(* IEC 61131-3 sources: Mizera_Tube/Plc (part 17) *)

*******************************************************************************
*   @@@ RICERCA BLOCCO
*******************************************************************************

LD   BUP_BLKSRC_PAGE               ** User in block search page
ST   GESTCH0.xBlkSearch

LD   %PLCFLAGS.1
ST   GESTCH0.xIntBlkSrc    * Forzam. esec. ricerca blocco interna

LD   %PlcOp0.2                     ** DryRun
ST   GESTCH0.xSpeedDryRunEnab ** Ab. velocita' di Dry Run (disabled in cnc.plc)

LD   %PLCFLAGS.0
ST   GESTCH0.xOverstore  * Ab. overstore dopo ricerca blocco (provv.)

LD   CondHoldCN0                   ** Condizioni richiesta hold canale 0
AND  PRGRUN_CN0                    ** M0.0 cn0.rc8.0  Programma in corso
ANDN BCO_CUSTOM_BOOT               ** rc8.18 Ciclo $BOOT in corso
ANDN BCO_CUSTOM_RESET              ** rc8.20 Ciclo $RESET in corso
ANDN PRGSTOP_CN0                   ** (cn0.rc8.1)  Programma interrotto CN0
ST   GESTCH0.xHold                * comando Hold al canale (esterno)

LD   Res_Ch0                       ** (gPlc25.3) reset channel 0
ST   GESTCH0.xReset               * comando RESET al canale (esterno)

CAL  FTRIG_POT (CLK:=Pon)          ** PON
CAL  TP_FTRIG_POT(IN:=FTRIG_POT.Q,PT:=300)

LD   %cn0.rc8.0
AND (
LD   bevAngleHead1_calc1                  * (C154) head 1 bevel angle
GE   70000
)
AND  %uvHeads0.uvhCommand[0].1          * UVH_COMMAND_PLC_VRTC_HANDLING
S    alarm_tool_surface

LD   %cn0.rc8.0
AND (
LD   %cn0.rc18                      * CO_ERRCODE
EQ   428                            * motion command error
)
S    alarm_motion_cmd_err

LD   Pul_Reset                     ** (gPlc0.3)Reset pushbutton
R    alarm_tool_surface
R    alarm_motion_cmd_err

LD   alarm_tool_surface
ST   %PLCerr4.0

LD   alarm_motion_cmd_err
ST   %PLCerr4.1

* todo CAL  RTRIG_TIPTOUCH(CLK:=%PLCerr5.4)

LD   Pul_Reset                     ** (gPlc0.3)Reset pushbutton
OR   Pul_Stop                      ** (gPlc0.2)Stop pushbutton
AND  ch0_in_ref                    ** channel 0 in ref
OR   EMER_GEN                      ** M0.10 Emergenza generale
***OR   LsrVrtcFcSoftware             ** (LsPlc0.31)Intervento Fc Sofware in lavorazione Laser
OR   TP_FTRIG_POT.Q
OR (
LD   %vrtc1.VrdwStatRegister1.2     * Upper mandatory position limit reached
OR   %vrtc1.VrdwStatRegister1.3     * Lower mandatory position limit reached
AND  %vrtc1.VrdwCtrlRegister0.1
)
* todo OR   RTRIG_TIPTOUCH.Q
OR   alarm_tool_surface
OR   alarm_motion_cmd_err
OR   Pul_Reset_EMERG                * Tasto RESET premuto per pi?di 4 secondi
ST   GESTCH0.xEmer

LD   ChannelFeedrate               ** feedrate for channel
ST   GESTCH0.xOverride
ST   AxesOverride

**********************************************************************
* Limitazione 10% to 100% in case of following supports in descending
**********************************************************************
LD   EnVSuppFeedRec
JMPCN STATE_EN_VSREC
LD   GESTCH0.xOverride
MULDIV(M=VSuppFeedReduction,D=1000)
ST   GESTCH0.xOverride
STATE_EN_VSREC:
**********************************************************************

CAL  GESTCH0

*******************************************************************************
*   @@@ RICERCA BLOCCO
*******************************************************************************
LD   GESTCH0.yBlkSearch
ST   BLKSRC_RUN                    ** Ricerca blocco in corso

LD   GESTCH0.yBlkSrcEnded * ricerca blocco terminata
ST   BLKSRC_END                    ** Ricerca blocco terminata

LD   0
ST   %cn0.BlkSearch.MskMoveA

LD   16#32
ST   %cn0.BlkSearch.Option

LD   BUP_BLKSRCPOINT               ** ui16.31 Ricerca blocco su punto intermedio
JMPCN INTPOINT

LD   16#72
ST   %cn0.BlkSearch.Option

INTPOINT:
LD   -1
ST   %ui6           ** Non generare M su overstore automatico
ST   %ui7           ** Non generare S/T su overstore automatico

***********************************************
* Gestione Informazioni per ripresa lavorazione
***********************************************

LD   Pul_Start                     ** (gPlc0.1)Start pushbutton
AND  ch0_in_aut                    ** channel 0 in aut
ANDN ExeAuxMode                    ** (gPlc0.29)Esecuzione ausiliaria 1000.PGM
S    MEM_INTPROG                   ** R15.0 Mem. programma valido per ripresa pezzo

LD   M30_CN0                       ** M0.13 M30:EndProgram CN0
ANDN ExeAuxMode                    ** (gPlc0.29)Esecuzione ausiliaria 1000.PGM
OR   BUP_PROGSEL                   ** ui16.30 Impulso selezione programma
R    MEM_INTPROG                   ** R15.0 Mem. programma valido per ripresa pezzo

* Lettura dati correnti durante esecuzione programma

LD   %cn0.rc8.0          * Programma in corso canale 0
ANDN %cn0.rc0.0          * Reset NC
***ANDN KeyStop_Tp          ** Stop level
ANDN %cn0.rc8.1          * rc8.1  Programma interrotto
ANDN %cn0.rc8.8
ANDN ExeAuxMode                    ** (gPlc0.29)Esecuzione ausiliaria 1000.PGM
JMPCN READ

LD   %cn0.lev0.curline
ST   CURRENT_LINE                  ** Numero riga corrente del part program in esecuzione

*******************************************
*   Calcola la posizione del TCP sul piano
*   della macchina
*******************************************
LDN  Gest5Ax                        ** (gPlc0.0)Gestione MAcchina 5 assi
JMPC Normal

LD   %ax0.ra54          ** X TCP
ST   locX                          ** Used in block search (ricerca blocco)

LD   %ax1.ra54          ** Y TCP
ST   locY                          ** Used in block search (ricerca blocco)

LD   %cn0.mat.sts0
EQ   16#B
JMPCN identity

LD   locX                          ** Used in block search (ricerca blocco)
DIV  100                ** DIV per problemi di overflow
MUL  %cn0.mat.a0
ADD  (
LD   locY                          ** Used in block search (ricerca blocco)
DIV  100
MUL  %cn0.mat.a1
)
DIV  10
ADD  (
LD   %cn0.mat.a3
DIV  1000
)
ST   XactualQta                    ** X actual quota Used in block search (ricerca blocco)

LD   locX                          ** Used in block search (ricerca blocco)
DIV  100                ** DIV per problemi di overflow
MUL  %cn0.mat.a4
ADD  (
LD   locY                          ** Used in block search (ricerca blocco)
DIV  100
MUL  %cn0.mat.a5
)
DIV  10
ADD  (
LD   %cn0.mat.a7
DIV  1000
)
ST   YactualQta                    ** Y actual quota Used in block search (ricerca blocco)

JMP  ComHead

identity:
LD   locX                          ** Used in block search (ricerca blocco)
ST   XactualQta                    ** X actual quota Used in block search (ricerca blocco)

LD   locY                          ** Used in block search (ricerca blocco)
ST   YactualQta                    ** Y actual quota Used in block search (ricerca blocco)

JMP  ComHead

Normal:
LD   %ax0.ra4           ** X
ST   XactualQta                    ** X actual quota Used in block search (ricerca blocco)

LD   %ax1.ra4           ** Y
ST   YactualQta                    ** Y actual quota Used in block search (ricerca blocco)

ComHead:
LD   XactualQta                    ** X actual quota Used in block search (ricerca blocco)
SUB  ORIGPRGX                      ** Origine programmata X
ST   MEM_XQUOTE                    ** R13 Memorizza quota X per collimazione ricerca blocco

LD   YactualQta                    ** Y actual quota Used in block search (ricerca blocco)
SUB  ORIGPRGY                      ** Origine programmata Y
ST   MEM_YQUOTE                    ** R14 Memorizza quota Y per collimazione ricerca blocco

READ:
* Azzera dati se programma non valido

LD   MEM_INTPROG                   ** R15.0 Mem. programma valido per ripresa pezzo
JMPC END_VALPR

LD   0
ST   CURRENT_LINE                  ** Numero riga corrente del part program in esecuzione
ST   MEM_XQUOTE                    ** R13 Memorizza quota X per collimazione ricerca blocco
ST   MEM_YQUOTE                    ** R14 Memorizza quota Y per collimazione ricerca blocco

END_VALPR:

* Passa i dati alla UI
* NB: occorre saltare l'aggiornamento nella modalita di overstore/auxcmd

LD   %cn0.rc8.26
ANDN %cn0.rc8.24
OR(
LD   %cn0.rc8.27
ANDN %cn0.rc8.25
)
JMPC OVERSTORERUN

LD   CURRENT_LINE                  ** Numero riga corrente del part program in esecuzione
*ADD  1
ST   PU_LASTLINE                   ** ui13 Ultima linea eseguita per ricerca blocco

LD   MEM_XQUOTE                    ** R13 Memorizza quota X per collimazione ricerca blocco
ST   PU_QCOLX                      ** ui2 Quota asse X collimazione ricerca blocco

LD   MEM_YQUOTE                    ** R14 Memorizza quota Y per collimazione ricerca blocco
ST   PU_QCOLY                      ** ui3 Quota asse Y collimazione ricerca blocco

OVERSTORERUN:

* Abilita quote per collimazione ricerca blocco

LD   MEM_INTPROG                   ** R15.0 Mem. programma valido per ripresa pezzo
ST   PLC_BPU_ENCOLDATA             ** ui0.31 Abilita quote per collimazione ricerca blocco

LD   PLC_BPU_ENCOLDATA             ** ui0.31 Abilita quote per collimazione ricerca blocco
ANDN PRGRUN_CN0                    ** M0.0 cn0.rc8.0  Programma in corso
ST   ResumeProgEnab                ** (gPlc25.0) Data avaiable for resume program

LD   Pul_Start                     ** (gPlc0.1)Start pushbutton
ANDN ExeAuxMode                    ** (gPlc0.29)Esecuzione ausiliaria 1000.PGM
AND  ch0_in_aut                    ** channel 0 in aut
S    BlackOut                      ** (R55.31)Interruzione per BlackOut

LD   FT_PRGRUN.Q        ** Dwn Programma in corso
OR   Pul_Reset                     ** (gPlc0.3)Reset pushbutton
OR   M30_CN0                       ** M0.13 M30:EndProgram CN0
R    BlackOut                      ** (R55.31)Interruzione per BlackOut

*******************************************************************************

LD   GESTCH0.yProgramRun * Programma in corso
ST   PRGRUN_CN0                    ** M0.0 cn0.rc8.0  Programma in corso

LD   BCO_STB_GET                   ** rc8.17 Strobe per GET resources
AND  AxStopSincGRP                 ** (gPlc13.11)Assi Fermi per sincronismo GRP[ax]
ST   BCI_ACK_GET                   ** rc0.29  ACK per GET resource

LD   GESTCH0.xRTPlus     * comando + in retrace
AND  %cn0.rc64.25        * Comando FWD Retrace
OR(
LD   GESTCH0.xRTMinus    * comando - in retrace
AND  %cn0.rc64.26        * Comando REV Retrace
)
AND  M_HOLD                        ** (gPlc19.0)Mem. Richiesta Hold
ST   Appoggio                      ** Appoggio

CAL  TOF_0(IN=Appoggio,PT=1000)    ** Appoggio

LD   TOF_0.Q
ST   RETRACERUN                    ** M0.11 Ciclo di retrace in Run

**************************
* FUNZIONI M DI SERVIZIO *
*      CANALE 0          *
**************************

LD   %rc9                * Registro funzioni M canale 0
EQ   10
AND  %rc8.4              * Strobe funzioni M canale 0
ST   M10_CN0                       ** M0.14 M10: Attiva Hold + Jog CN0

LD   %rc9                * Registro funzioni M canale 0
EQ   30
AND  %rc8.4              * Strobe funzioni M canale 0
ST   M30_CN0                       ** M0.13 M30:EndProgram CN0

LD   %rc9                * Registro funzioni M canale 0
EQ   2
AND  %rc8.4              * Strobe funzioni M canale 0
ST   M2_CN0                        ** M0.28 M2: EndProgram CN0 M2

LD   %rc9                * Registro funzioni M canale 0
EQ   32
AND  %rc8.4              * Strobe funzioni M canale 0
ST   M32TglMan                     ** M32: Attesa inizio taglio manuale

****************************************************************************************************

*** *** ***

LD   %rc9                * Registro funzioni M canale 0
EQ   600
AND  %rc8.4              * Strobe funzioni M canale 0
ST   M600_G81_84                   ** Richiesta Sblocco M40000_CN4: Richiesta Servizio per Unit_2]

CAL  TP_1(IN=M600_G81_84,PT=1000)  ** Impulso sblocco M40000

**************************
LD   %rc9                * Registro funzioni M canale 0
EQ   7000
AND  %rc8.4              * Strobe funzioni M canale 0
ST   M7000_RETR                    ** M7000: Retrace enable

LD   %rc9                * Registro funzioni M canale 0
EQ   8000
AND  %rc8.4              * Strobe funzioni M canale 0
ST   M8000_RETR                    ** M8000: Retrace disable
**************************

********************************************************************************
* DB Laser upload synchronism
********************************************************************************
*LD   %LSRPlcOp0.5                  ** Worklist mode enabled
*AND  %WlistMngt.wl_flag.0       ** Se codice DB gestito nella linea della lista di lavoro
*ORN  %LSRPlcOp0.5                  ** Worklist mode enabled
*JMPCN NoLoadDB

LD   %cn0.rc9                   ** Registro funzioni M canale 0
EQ   1000
AND  %cn0.rc8.4                 ** Strobe funzioni M canale 0
OR   isoLoadRecord                 ** (LsIso10.3) Load database record with Block search in run
ST   Up_Load_DB                    ** upload DB request

CAL  RTRIG_CAR_DB(CLK:=Up_Load_DB) ** Trig on upload DB request

LD   RTRIG_CAR_DB.Q
S    UpLoad_DB_Laser               ** (LsPlc0.0 )Comando Caricamento DataBase Laser

*NoLoadDB:
LD   FeedbackDBloaded              ** (LsGui1.0) upload DB request
OR   Pul_Reset                     ** (gPlc0.3)Reset pushbutton
OR   ON_ONE_SCAN                   ** PLCFLAGS.8  Flag on alla prima scansione PLC
R    UpLoad_DB_Laser               ** (LsPlc0.0 )Comando Caricamento DataBase Laser
R    isoLoadRecord                 ** (LsIso10.3) Load database record with Block search in run
R    Up_Load_DB                    ** upload DB request

***********************************************************************************

LD   %rc9                * Registro funzioni M canale 0
EQ   9999
AND  %rc8.4              * Strobe funzioni M canale 0
ST   M9999                         ** M9999: Abilitazione Start pae Canali Ausiliari

LD   M9999                         ** M9999: Abilitazione Start pae Canali Ausiliari
S    EabStartCnAux                 ** Abilitazione Start per canali ausiliari

LDN  PRGRUN_CN0                    ** M0.0 cn0.rc8.0  Programma in corso
OR   Res_Axes                      ** (gPlc25.1) reset axes disable electric shaft
R    EabStartCnAux                 ** Abilitazione Start per canali ausiliari

LD   M30_CN0                       ** M0.13 M30:EndProgram CN0
OR   M2_CN0                        ** M0.28 M2: EndProgram CN0 M2
S    PRGRUN_CN0_END                ** M0.4 Programma su canale 0 terminato con M30

LDN  PRGRUN_CN0                    ** M0.0 cn0.rc8.0  Programma in corso
ANDN PRGRUN_CN3                    ** M0.2 cn3.rc8.0  Programma in corso
R    PRGRUN_CN0_END                ** M0.4 Programma su canale 0 terminato con M30

* Sincronismo Richiesta servizio Da canale 0 a "Unit?Teste"
LD   %rc9                * Registro funzioni M canale 0
EQ   10000
AND  %rc8.4              * Strobe funzioni M canale 0
ANDN UnlockCn0funzReq              ** Sblocco richiesta servizio da CN0 [(M10000 iniziolav.) / M10001(finelav.)]
ST   M10000_CN0                    ** M0.8 M10000_CN0: Invoca Unit_1 (inizialavorazione)

LD   %rc9                * Registro funzioni M canale 0
EQ   10001
AND  %rc8.4              * Strobe funzioni M canale 0
AND  UnlockCn0funzReq              ** Sblocco richiesta servizio da CN0 [(M10000 iniziolav.) / M10001(finelav.)]
ST   M10001_CN0                    ** M0.9 M10001_CN0: Invoca Unit_1 (finelavorazione)

CAL R_TRIG10000(CLK=M10000_CN0)    ** M0.8 M10000_CN0: Invoca Unit_1 (inizialavorazione)
CAL R_TRIG10001(CLK=M10001_CN0)    ** M0.9 M10001_CN0: Invoca Unit_1 (finelavorazione)
CAL F_TRIG10000(CLK=M10000_CN0)    ** M0.8 M10000_CN0: Invoca Unit_1 (inizialavorazione)
CAL F_TRIG10001(CLK=M10001_CN0)    ** M0.9 M10001_CN0: Invoca Unit_1 (finelavorazione)

LD   R_TRIG10000.Q       ** FronteUp M10000_CN0: Invoca Unit_1 (inizialavorazione)
JMPCN INIZIOLAV
LD    1
ST   %FunzRequest                  ** Funzione richiesta per Unit_1
INIZIOLAV:

LD   R_TRIG10001.Q       ** Fronteup M10001_CN0: Invoca Unit_1 (finelavorazione)
JMPCN FINELAV
LD    2
ST   %FunzRequest                  ** Funzione richiesta per Unit_1
FINELAV:

LD   R_TRIG30000.Q       * FronteUp M30000_CN3: Attendi Servizio per Unit_1
OR   RT_PRGRUN.Q         ** Up Programma in corso
OR   FT_PRGRUN.Q         ** Dwn Programma in corso
JMPCN RESETVAL
LD   0
ST   %FunzRequest                  ** Funzione richiesta per Unit_1
RESETVAL:

**************************
* Attesa Start Con M10   *
**************************
CAL  RT_M10(CLK=M10_CN0)           ** M10: Attiva Hold + Jog

LD   RT_M10.Q            * M10: Attiva Hold + Jog
AND  AwaitStart                    ** Attesa Start
S    RestartOk                     ** Restart Ok (M10)

LD   RT_M10.Q            * M10: Attiva Hold + Jog
S    AwaitStart                    ** Attesa Start

LDN  M10_CN0                       ** M0.14 M10: Attiva Hold + Jog CN0
AND  RestartOk                     ** Restart Ok (M10)
ORN  %cn0.rc8.0          * Programma in corso
OR   Pul_Reset                     ** (gPlc0.3)Reset pushbutton
R    AwaitStart                    ** Attesa Start
R    RestartOk                     ** Restart Ok (M10)

******************************************************************
* FINE GESTIONE CANALE 0    -----------------------------------###
******************************************************************

LD   %cn3.cc1.2           * Maschera assi associata al canale 0
ANDN GESTAX29.yZeroed     * Asse tarato
AND  ch3_in_ref                    ** channel 3 in ref
ANDN PLC_SEL_SINGREF               ** ui16.28 Selezione REF singolo
ST   AxesHeadNoZeroed              ** Assi Testa non riferiti

******************************************************************************
*   GESTIONE LISTE DI LAVORO
*   (#WLIST)
******************************************************************************
LD   %LSRPlcOp0.5                  ** Worklist mode enabled
ST   WORK_LIST_MAIN.xEnable

LD   PRGRUN_CN0                    ** M0.0 cn0.rc8.0  Programma in corso
ST   WORK_LIST_MAIN.xProgRun

LD   LaserOn                       ** (LsPlc1.25) Per GUI  LaserOn
ST   WORK_LIST_MAIN.xEmissionOn

CAL  WORK_LIST_MAIN

******************************************************************************
* Allow general close loop timer

LD   TON_ABIL.Q          * Abilitazione drives
ANDN TOF_MALARM.Q        * Assi in allarme
ST   GeneralCloseLoop

******************************************************************************
*   GESTIONE ASSE VIRTUALE X
******************************************************************************
PATH %ax0

LD   %PLCFLAGS.0
ST   GESTAX0.xPlusLS     * Finecorsa +

LD   %PLCFLAGS.0
ST   GESTAX0.xMinusLS    * Finecorsa -

LD   TON_ABIL.Q          * Abilitazione drives
ANDN TOF_MALARM.Q        * Assi in allarme
AND  Pon                           ** PON
ST   GESTAX0.xCloseLoop

LD   %PLCFLAGS.0
ST   GESTAX0.xRefLS

*LD   %PLCFLAGS.0
*ST   GESTAX0.xSelected

LD   JOG_ENABLE                    ** (gPlc0.22)Jog Enable
AND  PRGSTOP_CN0                   ** (M0.27)  Programma interrotto CN0
AND  GESTAX27.xSelected
ST   GESTAX0.xSelected

LD   JOG_ENABLE                    ** (gPlc0.22)Jog Enable
AND  PRGSTOP_CN0                   ** (M0.27)  Programma interrotto CN0
AND  GESTAX27.xSelected
AND  %FUNCBTN.2
ST   GESTAX0.xJogPlus

LD   JOG_ENABLE                    ** (gPlc0.22)Jog Enable
AND  PRGSTOP_CN0                   ** (M0.27)  Programma interrotto CN0
AND  GESTAX27.xSelected
AND  %FUNCBTN.3
ST   GESTAX0.xJogMinus

LD   AxesHeadNoZeroed              ** Assi Testa non riferiti
OR   BlcAvX1_user                  ** M74.0 Blocco avanzamento asse X1 da user.plc
OR   CMD_HOLDMOVING_CH3.0          ** M202 Hold moving command axis CH3 (bit0=X, bit1=Y...)
ST   GESTAX0.xHoldMoving * Richiesta blocco avanzamento

LDN  ch0_in_ref                    ** channel 0 in ref
ST   GESTAX0.xEnFIR      * Abilita filtri FIR

LD   ALWAYS_ONE                    ** PLCFLAGS.1  Flag sempre stato on
ST   GESTAX0.xZeroForced * Forzamento asse tarato
ST   GESTAX0.xLockRef    * Blocco avvio ciclo REF da canale

*LD   %cn0.DisabVisAX.0
*ST   GESTAX0.xDisabVis    * Disabilita visualizzazone

CAL  GESTAX0

LD   JOGrunning                    ** One axis moving in JOG
OR   %ra19.1         * Stato JOG all'interno del canale
ST   JOGrunning                    ** One axis moving in JOG

LD   REFrunning                    ** One axis moving in REF
OR   %ra19.2
ST   REFrunning                    ** One axis moving in REF

LD   INCrunning                    ** One axis moving in INC
OR   %ra19.3
ST   INCrunning                    ** One axis moving in INC

LD   %pa9                * Velocit?massima asse
MUL  1000
DIV  60
ST   %ra50               * Limitazione velocita' massima interpolazione

LD   BSG_INC                       ** rg1.2 Selezione modo INC (inc.fissi)
JMPCN SVIX

LD   %pa59               * Velocit?di Repos
MUL  1000
DIV  60
MUL  AxesOverride                  ** (gPlc16) feed degli assi (%)
DIV  100
ST   %ra50               * Limitazione velocita' massima interpolazione

SVIX:

******************************************************************************
*   GESTIONE ASSE VIRTUALE Y
******************************************************************************
PATH %ax1

LD   %PLCFLAGS.0
ST   GESTAX1.xPlusLS     * Finecorsa +

LD   %PLCFLAGS.0
ST   GESTAX1.xMinusLS    * Finecorsa -

LD   TON_ABIL.Q          * Abilitazione drives
ANDN TOF_MALARM.Q        * Assi in allarme
AND  Pon                           ** PON
ST   GESTAX1.xCloseLoop

LD   %PLCFLAGS.0
ST   GESTAX1.xRefLS

LD   JOG_ENABLE                    ** (gPlc0.22)Jog Enable
AND  PRGSTOP_CN0                   ** (M0.27)  Programma interrotto CN0
AND  GESTAX28.xSelected
AND  %FUNCBTN.2
ST   GESTAX1.xJogPlus

LD   JOG_ENABLE                    ** (gPlc0.22)Jog Enable
AND  PRGSTOP_CN0                   ** (M0.27)  Programma interrotto CN0
AND  GESTAX28.xSelected
AND  %FUNCBTN.3
ST   GESTAX1.xJogMinus

*LD   %PLCFLAGS.0
*ST   GESTAX1.xSelected

LD   JOG_ENABLE                    ** (gPlc0.22)Jog Enable
AND  PRGSTOP_CN0                   ** (M0.27)  Programma interrotto CN0
AND  GESTAX28.xSelected
ST   GESTAX1.xSelected

LD   AxesHeadNoZeroed              ** Assi Testa non riferiti
OR   BlcAvY1_user                  ** M74.4 Blocco avanzamento asse Y da user.plc
OR   CMD_HOLDMOVING_CH3.1           ** M202 Hold moving command axis CH3 (bit0=X, bit1=Y...)
ST   GESTAX1.xHoldMoving * Richiesta blocco avanzamento

LDN  ch0_in_ref                    ** channel 0 in ref
ST   GESTAX1.xEnFIR      * Abilita filtri FIR

LD   ALWAYS_ONE                    ** PLCFLAGS.1  Flag sempre stato on
ST   GESTAX1.xZeroForced * Forzamento asse tarato
ST   GESTAX1.xLockRef    * Blocco avvio ciclo REF da canale

CAL  GESTAX1

LD   JOGrunning                    ** One axis moving in JOG
OR   %ra19.1         * Stato JOG all'interno del canale
ST   JOGrunning                    ** One axis moving in JOG

LD   REFrunning                    ** One axis moving in REF
OR   %ra19.2
ST   REFrunning                    ** One axis moving in REF

LD   INCrunning                    ** One axis moving in INC
OR   %ra19.3
ST   INCrunning                    ** One axis moving in INC

LD   %pa9                * Velocit?massima asse
MUL  1000
DIV  60
ST   %ra50               * Limitazione velocita' massima interpolazione

LD   BSG_INC                       ** rg1.2 Selezione modo INC (inc.fissi)
JMPCN SVIY

LD   %pa59               * Velocit?di Repos
MUL  1000
DIV  60
MUL  AxesOverride                  ** (gPlc16) feed degli assi (%)
DIV  100
ST   %ra50               * Limitazione velocita' massima interpolazione

SVIY:

******************************************************************************
*   GESTIONE ASSE VIRTUALE Z
******************************************************************************
LD  %cn0.cc1.2           * Maschera assi associata al canale 0
JMPCN NOAX2

PATH %ax2

LD   %PLCFLAGS.0         * Flag sempre stato on
ST   GESTAX2.xPlusLS     * Finecorsa +

LD   %PLCFLAGS.0         * Flag sempre stato on
ST   GESTAX2.xMinusLS    * Finecorsa -

LD   TON_ABIL.Q          * Abilitazione drives
ANDN TOF_MALARM.Q        * Assi in allarme
AND  Pon                           ** PON
ST   GESTAX2.xCloseLoop

LD   %PLCFLAGS.0         * Flag sempre stato off
ST   GESTAX2.xRefLS

LD   %PLCFLAGS.0
ST   GESTAX2.xSelected

LD   ALWAYS_ONE
ST   GESTAX2.xDisLimiter

LD   %PLCerr5.4      **PLC Err 164 Tip touch (A11=1, A14=0, A15=0 in normal operation)
AND  ax2_Commanded                 ** %ax2.ra3.13 Axis 2 commanded to moving
ANDN ax2_GoFordward                ** %ax2.ra3.2 Axis 2 moving to positive
OR   CMD_HOLDMOVING_CH3.2          ** M202 Hold moving command axis CH3 (bit0=X, bit1=Y...)
***OR   JogCommandTipTouch
ST   GESTAX2.xHoldMoving * Richiesta blocco avanzamento
ST   GESTAX2_xHoldMoving

LDN  ch0_in_ref                    ** channel 0 in ref
ANDN DisabFir_CH0_axes.2
ST   GESTAX2.xEnFIR      * Abilita filtri FIR

LD   ALWAYS_ONE                    ** PLCFLAGS.1  Flag sempre stato on
ST   GESTAX2.xZeroForced * Forzamento asse tarato
ST   GESTAX2.xLockRef    * Blocco avvio ciclo REF da canale

CAL  GESTAX2

LD   JOGrunning                    ** One axis moving in JOG
OR   %ra19.1         * Stato JOG all'interno del canale
ST   JOGrunning                    ** One axis moving in JOG

LD   REFrunning                    ** One axis moving in REF
OR   %ra19.2
ST   REFrunning                    ** One axis moving in REF

LD   INCrunning                    ** One axis moving in INC
OR   %ra19.3
ST   INCrunning                    ** One axis moving in INC

LD   %pa9                * Velocit?massima asse
MUL  1000
DIV  60
ST   %ra50               * Limitazione velocita' massima interpolazione

LD   %vrtc5.VrdwCtrlRegister0.18 * De overlap
JMPCN NOAX2

LD   0
ST   %ra50               * Limitazione velocita' massima interpolazione

NOAX2:

******************************************************************************
*   GESTIONE ASSE VIRTUALE U
******************************************************************************
LD   %cn0.cc1.3           * Maschera assi associata al canale 0
JMPCN NO_U

PATH %ax6

LD   %PLCFLAGS.0
ST   GESTAX6.xPlusLS     * Finecorsa +

LD   %PLCFLAGS.0
ST   GESTAX6.xMinusLS    * Finecorsa -

LD   TON_ABIL.Q          * Abilitazione drives
ANDN TOF_MALARM.Q        * Assi in allarme
AND  Pon                           ** PON
ST   GESTAX6.xCloseLoop

LD   %PLCFLAGS.0
ST   GESTAX6.xRefLS

LD   %PLCFLAGS.0
ST   GESTAX6.xSelected

LD   AxesHeadNoZeroed              ** Assi Testa non riferiti
OR   BlcAvX1_user                  ** M74.0 Blocco avanzamento asse X1 da user.plc
OR   CMD_HOLDMOVING_CH3.3            ** M202 Hold moving command axis CH3 (bit0=X, bit1=Y...)
ST   GESTAX6.xHoldMoving * Richiesta blocco avanzamento

LD   ALWAYS_ONE                    ** PLCFLAGS.1  Flag sempre stato on
ST   GESTAX6.xZeroForced * Forzamento asse tarato
ST   GESTAX6.xLockRef    * Blocco avvio ciclo REF da canale

LD   %PLCFLAGS.0
ST   GESTAX6.xFromPlc

LDN  ch0_in_ref                    ** channel 0 in ref
ST   GESTAX6.xEnFIR      * Abilita filtri FIR

CAL  GESTAX6

LD   JOGrunning                    ** One axis moving in JOG
OR   %ra19.1         * Stato JOG all'interno del canale
ST   JOGrunning                    ** One axis moving in JOG

LD   REFrunning                    ** One axis moving in REF
OR   %ra19.2
ST   REFrunning                    ** One axis moving in REF

LD   INCrunning                    ** One axis moving in INC
OR   %ra19.3
ST   INCrunning                    ** One axis moving in INC
NO_U:

******************************************************************************
*   GESTIONE ASSE VIRTUALE V
******************************************************************************
LD   %cn0.cc1.4           * Maschera assi associata al canale 0
JMPCN NO_V

PATH %ax7

LD   %PLCFLAGS.0
ST   GESTAX7.xPlusLS     * Finecorsa +

LD   %PLCFLAGS.0
ST   GESTAX7.xMinusLS    * Finecorsa -

LD   TON_ABIL.Q          * Abilitazione drives
ANDN TOF_MALARM.Q        * Assi in allarme
AND  Pon                           ** PON
ST   GESTAX7.xCloseLoop

LD   %PLCFLAGS.0
ST   GESTAX7.xRefLS

LD   %PLCFLAGS.0
ST   GESTAX7.xSelected

LD   AxesHeadNoZeroed              ** Assi Testa non riferiti
OR   BlcAvX1_user                  ** M74.0 Blocco avanzamento asse X1 da user.plc
OR   CMD_HOLDMOVING_CH3.4            ** M202 Hold moving command axis CH3 (bit0=X, bit1=Y...)
ST   GESTAX7.xHoldMoving * Richiesta blocco avanzamento

LD   ALWAYS_ONE                    ** PLCFLAGS.1  Flag sempre stato on
ST   GESTAX7.xZeroForced * Forzamento asse tarato
ST   GESTAX7.xLockRef    * Blocco avvio ciclo REF da canale

LD   %PLCFLAGS.0
ST   GESTAX7.xFromPlc

LDN  ch0_in_ref                    ** channel 0 in ref
ST   GESTAX7.xEnFIR      * Abilita filtri FIR

CAL  GESTAX7

LD   JOGrunning                    ** One axis moving in JOG
OR   %ra19.1         * Stato JOG all'interno del canale
ST   JOGrunning                    ** One axis moving in JOG

LD   REFrunning                    ** One axis moving in REF
OR   %ra19.2
ST   REFrunning                    ** One axis moving in REF

LD   INCrunning                    ** One axis moving in INC
OR   %ra19.3
ST   INCrunning                    ** One axis moving in INC
NO_V:

******************************************************************************
*   GESTIONE ASSE REALE W (FOCALE)
******************************************************************************
LD   %ax9.ra83.4                   * PON Assi
OR   %ax9.pa3.31                   * Simulato
ORN  %cn0.cc1.5                    * Maschera assi associata al canale 0 W
OR(
LD   %nvel11            ** 3,4=CANopen, Ecat
EQ   3
)
OR(
LD   %nvel11            ** 3,4=CANopen, Ecat
EQ   4
)
OR   (
LD   I_I_READY_DRIVE_W             ** Ready signal drive W (external focal)
AND  (
LD   %ax9.nvel11
EQ   0
)
)
ST   Pon_WLens                     ** PON Axe W_Lens

LD  %cn0.cc1.5                     * Maschera assi associata al canale 0 W
JMPCN NOAX9

PATH %ax9
PATH %ax_lsref9

LD   %lsrefmode
ST   AXLSREF9.x_REF_mode        * 0=use ref switch...

LD   %lsreflevel
ST   AXLSREF9.x_TYPE_LS         * (1=NC, 0=NO)

LD   I_I_FC_W1_NEG                 ** W minimumm limit switch
ST   AXLSREF9.x_MIN_LS          * Min Limit switch

LD   I_I_FC_W1_POS                 ** W maximun limit switch
ST   AXLSREF9.x_MAX_LS          * Max Limit switch

*LD   I_I_INDEX_W1                  ** W1 Axis Homing Switch
LD   ALWAYS_ZERO
ST   AXLSREF9.x_REF_S           * Reference switch

CAL  AXLSREF9

LD   AXLSREF9.y_MIN_LS          * Min Limit switch
ST   GESTAX9.xMinusLS           * Negative limit switch

LD   AXLSREF9.y_MAX_LS          * Max Limit switch
ST   GESTAX9.xPlusLS            * Positive limit switch

LD   AXLSREF9.y_REF_S           * Reference switch
ST   GESTAX9.xRefLS             * Reference

LD   TON_ABIL.Q                    * Abilitazione drives
ANDN TOF_MALARM.Q                  * Assi in allarme
AND  Pon                           ** PON
ST   GESTAX9.xCloseLoop

LD   SelManAxe_Lens                ** (gGui0.14)Selezione W_Lens -
OR   (
LD   GSTMAC.yChSelMask.0
AND  SEL_ASSE.yExtMask.5
)
ANDN PRGRUN_CN0                    ** M0.0 cn0.rc8.0  Programma in corso
ST   GESTAX9.xSelected

LD   WLensplus                     ** (gGui0.12)Comando W_Lens +
AND  EnabJogRTCP                   ** Abilita Jog RTCP
AND  SelManAxe_Lens                ** (gGui0.14)Selezione W_Lens -
ANDN PRGRUN_CN0                    ** M0.0 cn0.rc8.0  Programma in corso
OR   WLensplus                     ** (gGui0.12)Comando W_Lens +
ST   GESTAX9.xJogPlus

LD   WLensmimus                    ** (gGui0.13)Comando W_Lens -
AND  EnabJogRTCP                   ** Abilita Jog RTCP
AND  SelManAxe_Lens                ** (gGui0.14)Selezione W_Lens -
ANDN PRGRUN_CN0                    ** M0.0 cn0.rc8.0  Programma in corso
OR   WLensmimus                    ** (gGui0.13)Comando W_Lens -
ST   GESTAX9.xJogMinus

LDN  ch0_in_ref                    ** channel 0 in ref
ANDN EnJogRtcp                     ** (gPlc0.18)Abilitazione Jog RTCP tuning
ST   GESTAX9.xEnFIR               * Abilita filtri FIR
ST   GESTAX9.xEnFrComp            ** Abilita friction compensation

LD   ALWAYS_ZERO                   ** PLCFLAGS.0  Flag sempre stato off
ST   GESTAX9.xDisLimiter

*LD   CMD_HOLDMOVING_CH3.5          ** M202 Hold moving command axis CH3 (bit0=X, bit1=Y...)
LD   ALWAYS_ZERO
ST   GESTAX9.xHoldMoving          * Richiesta blocco avanzamento

CAL  TOF_GRANT_AX9 (IN:=Res_Axes,PT:=300) ** (gPlc25.1) reset axes disable electric shaft

LD   %cn0.rc8.2  *BCO_CANREADY        * rc8.2  Canale Ready
ANDN %ra3.15   *BAO_ALLM            * ra3.15  Asse in Allarme
ANDN ch0_in_ref                    ** channel 0 in ref
ANDN BUP_JOGOPEN                   ** ui16.16 Selezione esecuzione JOG a loop aperto
ANDN TOF_GRANT_AX9.Q
ST   GESTAX9.xFromPlc

*POSITIONING
    *{
        LD   %nvel11             * PAR-PLC tipo di drive, 4=Canopen positioning
        EQ   4
        JMPCN END_PREGESTAX_POSITIONINGA

        LD   %cn0.rc8.2  *BCO_CANREADY        * rc8.2  Canale Ready
        ANDN %ra3.15   *BAO_ALLM            * ra3.15  Asse in Allarme
        AND(
        LD   AX9_CAN.yax_BUSY
        OR   AX9_CAN_AUX.yax_BUSY
        ANDN %ra0.15   *BAI_RESALARM        * ra0.15 Ripristino allarme asse
        ORN  %pa3.31    *AP_OPZIONI31        * pa3.31 Asse in simulato
        OR   PRGRUN_CN0                    ** M0.0 cn0.rc8.0  Programma in corso
        )
        ST   GESTAX9.xFromPlc

        END_PREGESTAX_POSITIONINGA:

        LD    100
        ST    %ra1
    *}

LD   %PLCFLAGS.0
ST   GESTAX9.xZeroForced          * Forzamento asse tarato
ST   GESTAX9.xLockRef             * Blocco avvio ciclo REF da canale

LD   Res_Axes                      ** (gPlc25.1) reset axes disable electric shaft
ST   GESTAX9.xUnlock

LD   %cn0.rc8.3            * ch0 in alarm
OR   %cn3.rc8.3            * ch3 in alarm
ST   GESTAX9.xSetAlarm     ** Forzamento allarme asse

CAL  GESTAX9

LD   JOGrunning                    ** One axis moving in JOG
OR   %ra19.1         * Stato JOG all'interno del canale
ST   JOGrunning                    ** One axis moving in JOG

LD   REFrunning                    ** One axis moving in REF
OR   %ra19.2
ST   REFrunning                    ** One axis moving in REF

LD   INCrunning                    ** One axis moving in INC
OR   %ra19.3
ST   INCrunning                    ** One axis moving in INC

LD   GESTAX9.yDriveNotEn
ST   %PLCerr2.7                    * Axis 9, drive not enable

*--------- POSITIONING
  LD   %nvel11             * PAR-PLC tipo di drive, 4=Canopen positioning
  EQ   4
  JMPCN END_POSTGESTAX_POSITIONINGA

  LD   %rc8.2              * CN-PLC Canale Ready
  ANDN %rc0.1              * Emergenza dal canale agli assi
  ANDN %rc0.0              * PLC-CN Reset CN canale
  ST   AX9_CAN.xax_ENABLE
  ST   AX9_CAN_AUX.xax_ENABLE

  CAL  AX9_CAN

  CAL  AX9_CAN_AUX

END_POSTGESTAX_POSITIONINGA:
*--------- POSITIONING

LD   %pa9                          * Velocit?massima asse
MUL  1000
DIV  60
ST   %ra50                         * Limitazione velocita' massima interpolazione

LD   %vrtc5.VrdwCtrlRegister0.18   * De overlap
JMPCN NOAX9BIS
LD   0
ST   %ra50                         * Limitazione velocita' massima interpolazione
NOAX9BIS:

LD   StartPosFocale                ** (LsIso86) Comando Posizione Focale
ORN  PRGRUN_CN0                    ** M0.0 cn0.rc8.0  Programma in corso
R    LensPosEnd                    ** (LsPlc63.0) Lens positioning finish

CAL  TRIG_MOV_REQ (CLK:=PulsMoveFocal) ** (LsGui1.5) Focal command to move to set point
CAL  RTRIG_MOVE_REM_CONTR(CLK:=RemContrFoc0) ** Xhc_Puls.30 Move focal at 0 mm      *

LD   TRIG_MOV_REQ.Q
S    MoveByUser

LD   RTRIG_MOVE_REM_CONTR.Q
S    MoveAtZero                    ** Remote controller command

LD   StartPosFocale                ** (LsIso86) Comando Posizione Focale
OR   MoveByUser
OR   MoveAtZero                    ** Remote controller command
ST   POS_AX9.xax_ENABLE

LDN  POS_AX9.xax_ENABLE
ST   POS_AX9.xax_CLEAR

LD   POS_AX9.xax_ENABLE
AND  POS_AX9.yax_READY
ANDN POS_AX9.yax_ENDOK
ANDN POS_AX9.yax_ENDERR
ST   POS_AX9.xax_START

LD   %TabLsr0.L_CutFocal                   ** Valore focale passato da tabelle
ST   temp

***************************************
*   Focal=funz(angle)
*   #CDL
***************************************
LD   PRGRUN_CN0
ANDN PRGSTOP_CN0
AND (
LD   %uvHeads0.uvhCommand1
EQ   4                              * Cutting phase
)
AND  %LSRPlcOp0.3
JMPCN no_corr_focal
     LD   temp
     ADD (
     LD   temp
     MULDIV(M=%TsCutDataLinear.CDL_Focal,D=100000) * 100 %
     )
     ST   temp
no_corr_focal:

LD   PRGRUN_CN0                    ** M0.0 cn0.rc8.0  Programma in corso
JMPCN focal_by_program
     LD   temp
     ST   POS_AX9.xax_QUOTA
focal_by_program:

LDN  PRGRUN_CN0                    ** M0.0 cn0.rc8.0  Programma in corso
JMPCN focal_by_user
LD   FocByUser                     ** (LsGui74) Set-point for focal movement by user
ST   POS_AX9.xax_QUOTA

LD   MoveAtZero                    ** Remote controller command
JMPCN no_0
LD   0
ST   POS_AX9.xax_QUOTA
no_0:
focal_by_user:

LD   %pa9
ST   POS_AX9.xax_VEL

CAL  POS_AX9

LD   POS_AX9.yax_ENDOK
S    LensPosEnd                    ** (LsPlc63.0) Lens positioning finish

LD   %ax9.ra4
DIV  10
EQ (
LD   FocByUser                     ** (LsGui74) Set-point for focal movement by user
DIV  10
)
OR   Pul_Reset                     ** (gPlc0.3)Reset pushbutton
OR   I_I_EMERGENZA                 ** Machine OK (no EMERG.)
OR   EMER_GEN                      ** M0.10 Emergenza generale
OR   Pul_Start                     ** (gPlc0.1)Start pushbutton
R    MoveByUser

LD   MoveAtZero                    ** Remote controller command
AND  (
LD   %ax9.ra4
DIV  10
EQ   0
)
OR   Pul_Reset                     ** (gPlc0.3)Reset pushbutton
OR   I_I_EMERGENZA                 ** Machine OK (no EMERG.)
OR   EMER_GEN                      ** M0.10 Emergenza generale
OR   Pul_Start                     ** (gPlc0.1)Start pushbutton
R    MoveAtZero                    ** Remote controller command

LD   POS_AX9.yax_ENDOK
ORN  PRGRUN_CN0                    ** M0.0 cn0.rc8.0  Programma in corso
ST   appoggio                      ** Appoggio

CAL  RTRIG_RES_FOC (CLK:=appoggio) ** Appoggio

LD   RTRIG_RES_FOC.Q
JMPCN no_res_word
LD    ALWAYS_ZERO                  ** PLCFLAGS.0  Flag sempre stato off
ST    StartPosFocale               ** (LsIso86) Comando Posizione Focale
no_res_word:

NOAX9:

******************************************************************************
*   GESTIONE ASSE VIRTUALE A (HEAD)
******************************************************************************
LD   %cn0.cc1.6           * Maschera assi associata al canale 0
JMPCN NO_A

PATH %ax3

LD   %PLCFLAGS.0
ST   GESTAX3.xPlusLS     * Finecorsa +

LD   %PLCFLAGS.0
ST   GESTAX3.xMinusLS    * Finecorsa -

LD   TON_ABIL.Q          * Abilitazione drives
ANDN TOF_MALARM.Q        * Assi in allarme
AND  Pon                           ** PON
ST   GESTAX3.xCloseLoop

LD   %PLCFLAGS.0
ST   GESTAX3.xSelected

LD   AxesHeadNoZeroed              ** Assi Testa non riferiti
OR   BlcAvX1_user                  ** M74.0 Blocco avanzamento asse X1 da user.plc
OR   BlcAvY1_user                  ** M74.4 Blocco avanzamento asse Y da user.plc
OR   CMD_HOLDMOVING_CH3.6          ** M202 Hold moving command axis CH3 (bit0=X, bit1=Y...)
ST   GESTAX3.xHoldMoving * Richiesta blocco avanzamento

LDN  ch0_in_ref                    ** channel 0 in ref
ST   GESTAX3.xEnFIR      * Abilita filtri FIR

LD   %PLCFLAGS.0         * Flag sempre stato off
ST   GESTAX3.xRefLS

LD   ALWAYS_ONE                    ** PLCFLAGS.1  Flag sempre stato on
ST   GESTAX3.xLockRef    * Blocco avvio ciclo REF da canale
ST   GESTAX3.xZeroForced * Forzamento asse tarato

CAL  GESTAX3

LD   JOGrunning                    ** One axis moving in JOG
OR   %ra19.1         * Stato JOG all'interno del canale
ST   JOGrunning                    ** One axis moving in JOG

LD   REFrunning                    ** One axis moving in REF
OR   %ra19.2
ST   REFrunning                    ** One axis moving in REF

LD   INCrunning                    ** One axis moving in INC
OR   %ra19.3
ST   INCrunning                    ** One axis moving in INC

NO_A:

******************************************************************************
*   GESTIONE ASSE VIRTUALE B (HEAD)
******************************************************************************
LD  %cn0.cc1.7           * Maschera assi associata al canale 0
JMPCN NO_B

PATH %ax4

LD   %PLCFLAGS.0
ST   GESTAX4.xPlusLS     * Finecorsa +

LD   %PLCFLAGS.0
ST   GESTAX4.xMinusLS    * Finecorsa -

LD   TON_ABIL.Q          * Abilitazione drives
ANDN TOF_MALARM.Q        * Assi in allarme
AND  Pon                           ** PON
ST   GESTAX4.xCloseLoop

LD   %PLCFLAGS.0
ST   GESTAX4.xRefLS

LD   ALWAYS_ONE                    ** PLCFLAGS.1  Flag sempre stato on
ST   GESTAX4.xLockRef    * Blocco avvio ciclo REF da canale
ST   GESTAX4.xZeroForced * Forzamento asse tarato

LD   %PLCFLAGS.0
ST   GESTAX4.xSelected

LD   AxesHeadNoZeroed              ** Assi Testa non riferiti
OR   BlcAvX1_user                  ** M74.0 Blocco avanzamento asse X1 da user.plc
OR   BlcAvY1_user                  ** M74.4 Blocco avanzamento asse Y da user.plc
OR   CMD_HOLDMOVING_CH3.7          ** M202 Hold moving command axis CH3 (bit0=X, bit1=Y...)
ST   GESTAX4.xHoldMoving * Richiesta blocco avanzamento

LD   %PLCFLAGS.0
ST   GESTAX4.xFromPlc

LDN  ch0_in_ref                    ** channel 0 in ref
ST   GESTAX4.xEnFIR      * Abilita filtri FIR

CAL  GESTAX4

LD   JOGrunning                    ** One axis moving in JOG
OR   %ra19.1         * Stato JOG all'interno del canale
ST   JOGrunning                    ** One axis moving in JOG

LD   REFrunning                    ** One axis moving in REF
OR   %ra19.2
ST   REFrunning                    ** One axis moving in REF

LD   INCrunning                    ** One axis moving in INC
OR   %ra19.3
ST   INCrunning                    ** One axis moving in INC

NO_B:

******************************************************************************
*   GESTIONE ASSE VIRTUALE C (HEAD)
******************************************************************************
LD   %cn0.cc1.8           * Maschera assi associata al canale 0
JMPCN NO_C

PATH %ax5

LD   %PLCFLAGS.0
ST   GESTAX5.xPlusLS     * Finecorsa +

LD   %PLCFLAGS.0
ST   GESTAX5.xMinusLS    * Finecorsa -

LD   TON_ABIL.Q          * Abilitazione drives
ANDN TOF_MALARM.Q        * Assi in allarme
AND  Pon                           ** PON
ST   GESTAX5.xCloseLoop

LD   %PLCFLAGS.0
ST   GESTAX5.xRefLS

LD   %PLCFLAGS.0
ST   GESTAX5.xSelected

LDN  GESTAX2.yZeroed     * Asse tarato
AND  %cn0.cc1.2           * Maschera assi associata al canale 0
ORN  GESTAX1.yZeroed     * Asse tarato
AND  ch0_in_ref                    ** channel 0 in ref
ANDN %ui16.28            * Selezione Ref Singolo da UI
OR   CMD_HOLDMOVING_CH3.8            ** M202 Hold moving command axis CH3 (bit0=X, bit1=Y...)
OR   CMD_HOLDMOVING_CH5.8          ** M203 Hold moving command axis CH5 (bit0=X, bit1=Y...)
ST   GESTAX5.xHoldMoving * Richiesta blocco avanzamento

LD   ALWAYS_ONE                    ** PLCFLAGS.1  Flag sempre stato on
ST   GESTAX5.xZeroForced * Forzamento asse tarato
ST   GESTAX5.xLockRef    * Blocco avvio ciclo REF da canale

LD   %PLCFLAGS.0
ST   GESTAX5.xFromPlc

LDN  ch0_in_ref                    ** channel 0 in ref
ST   GESTAX5.xEnFIR      * Abilita filtri FIR

LD   ALWAYS_ONE
ST   GESTAX5.xDisLimiter      * Abilita filtri FIR

CAL  GESTAX5

LD   JOGrunning                    ** One axis moving in JOG
OR   %ra19.1         * Stato JOG all'interno del canale
ST   JOGrunning                    ** One axis moving in JOG

LD   REFrunning                    ** One axis moving in REF
OR   %ra19.2
ST   REFrunning                    ** One axis moving in REF

LD   INCrunning                    ** One axis moving in INC
OR   %ra19.3
ST   INCrunning                    ** One axis moving in INC

NO_C:

****************************************************************************************************
* Asse S (Mandrino) ----------------------------------------------------
****************************************************************************************************
PATH %ax10

LD   %ax10.ra83.4                  * PON Assi
OR   %ax10.pa3.31                  * Simulato
ORN  %cn0.cc1.9                    * Maschera assi associata al canale 0 S
ST   Pon_Mand                      ** PON Axe Mandrino

* GESTIONE MANDRINO CON ENCODER -----------------------------------------------

LD   %cn0.cc1.9                    * Maschera assi associata al canale 0
JMPCN NOMAND

LD   %PLCFLAGS.0
ST   GESTMAND.xM5Force             * Funzione M5 forzata

LD   ALWAYS_ONE                    ** PLCFLAGS.1  Flag sempre stato on
ST   GESTMAND.xSelFromInput        * Disabilita selezioni standard macchina

LD   100
ST   GESTMAND.xOverride            * override mandrino

LD   I_I_INDEX_MAND                *(IW4.1) CHUCK Axis Homing Switch
ST   GESTMAND.xRefLS

LDN  EMER_GEN
ST   GESTMAND.xRotatEnab

LD   %PLCFLAGS.1
ST   SICROTJOG                     ** rgc0.13 Sic. da revolver per rotazione mandrino in JOG

LD   I_I_CW
OR   I_I_CCW
ST   SelForaS                      ** (gPlc13.25)Selezione Asse S da Pagina Foratrice selezionata

LD   GSTMAC.yChSelMask.0
AND  SEL_ASSE.yExtMask.9           * canale X selezionato
OR   SelForaS                      ** (gPlc13.25)Selezione Asse S da Pagina Foratrice selezionata
ST   GESTMAND.xSelected

LD   Pul_Jogp                      ** Jog+ pushbutton (Ch0)
OR   I_I_CW
AND  GESTMAND.xSelected
AND  GESTMAND.xRotatEnab
ST   GESTMAND.xJogPlus             * Comando manuale avanti

LD   Pul_Jogm                      ** Jog- pushbutton (Ch0)
OR   I_I_CCW
AND  GESTMAND.xSelected
AND  GESTMAND.xRotatEnab
ST   GESTMAND.xJogMinus            * Comando manuale indietro

CAL  GESTMAND

*LD   GESTMAND.yErrOrienta
*ST   Plcerr  ** (C51.14) Error in Spindle Orientation request

***  yOkRpm: BOOL; * Mandrino a regime
***  yStopped: BOOL; * Mandrino fermo(ra3.0)
***  yZeroed: BOOL; * Mandrino tarato(ra3.14)
***  yInAlarm: BOOL; * Mandrino in allarme

NOMAND:

* Ack Funzioni M Canale 0 -------------------------------------------------------------
LDN  RestartOk                     ** Restart Ok (M10)
AND  M10_CN0                       ** M0.14 M10: Attiva Hold + Jog CN0
OR(
LD   M600_G81_84                   ** Richiesta Sblocco M40000_CN4: Richiesta Servizio per Unit_2]
AND  M40000_CN4                    ** (gPlc0.8)M40000_CN4: Attendi Servizio per Unit_2[]
)
OR   M10000_CN0                    ** M0.8 M10000_CN0: Invoca Unit_1 (inizialavorazione)
OR   M10001_CN0                    ** M0.9 M10001_CN0: Invoca Unit_1 (finelavorazione)
OR   GESTCH0.yWaitMFun
OR   (
LD   Up_Load_DB                    ** upload DB request
ANDN FeedbackDBloaded              ** (LsGui1.0) upload DB request
)
OR   WaitMfunc0Usr                 ** wait m function on ch0
OR   Ack_Mfun_PLC                  ** (gPlc0.11)Sblocco funzioni M da PLC.plc
OR   Ack_Mfun_UsrM                 ** (gPlc13.13) Unlock M-Functions from User_M
OR   WaitGasFlow                   ** (C56.0) M function iso wait
OR   SPURGOrun                     ** M107.2 Gas purge in progress
OR   M30_CN0                       ** M0.13 M30:EndProgram CN0
OR   M2_CN0                        ** M0.28 M2: EndProgram CN0 M2
ST   CH0END.xWaitMFun

CAL  CH0END

*******************************************************************************
*******************************************************************************
*   @@@ CH3 TESTA 1
*******************************************************************************
*******************************************************************************
PATH %cn3

LD   ALWAYS_ONE                    ** PLCFLAGS.1  Flag sempre stato on
ST   GESTCH3.xCmdFromInput

LD   ALWAYS_ONE                    ** PLCFLAGS.1  Flag sempre stato on
ST   GESTCH3.xEscOpCmd

LD   %PLCFLAGS.0
ST   GESTCH3.xSelFromInput        * Disabilita selezioni standard macchina

LD   Op_Mode0.ySelRef
ST   GESTCH3.xSelREF

LD   Op_Mode0.ySelSingRef
ST   GESTCH0.xSingleRef

LD   Op_Mode0.ySelJog
OR   JOG_ENABLE
ST   GESTCH3.xSelJOG

LD   Op_Mode0.ySelInc
ST   GESTCH3.xSelINC

LD   Op_Mode0.ySelMdi
* todo
*AND (
*LD   UP_SELCHAN                    ** ui17 Canale selezionato da monitor canale
*EQ   3
*)
ST   GESTCH3.xSelMDI

LD   Op_Mode0.ySelAut
ST   GESTCH3.xSelAUT

LD   PRGRUN_CN0                    ** M0.0 cn0.rc8.0  Programma in corso
ANDN PRGRUN_CN3                    ** M0.2 cn3.rc8.0  Programma in corso
OR(
LD   Pul_Start                     ** (gPlc0.1)Start pushbutton
AND  BCO_PRGRUN                    ** rc8.0  Programma in corso
AND  BCO_PRGINT                    ** rc8.1  Programma interrotto
)
AND  EabStartCnAux                 ** Abilitazione Start per canali ausiliari
ANDN GSTMAC.xReset
ANDN TOF_RESET.Q                    * Reset execution
OR   (
LD   GESTCH0.xStart
AND  %cn0.rc0.8
)
OR(
LD   Pul_Start                     ** (gPlc0.1)Start pushbutton
AND  BCI_MDI                       ** rc0.11  Selettore modi operativi su MDI (semiautom)
AND (
 LD   UP_SELCHAN                    ** ui17 Canale selezionato da monitor canale
 EQ   3
)
ANDN EMER_GEN                      ** M0.10 Emergenza generale
)
OR(
LD   StartAftTipTouch
ANDN EMER_GEN
ANDN GSTMAC.xReset
ANDN TOF_RESET.Q
)
ST   GESTCH3.xStart                 * comando START al canale (esterno)

LD   Res_Ch3                       ** (gPlc25.2) reset channel 3
ST   GESTCH3.xReset               * comando RESET al canale (esterno)

LD   CondHoldCN0                   ** Condizioni richiesta hold canale 0
OR(
LD   Pul_Stop                      ** (gPlc0.2)Stop pushbutton
AND  BCI_MDI                       ** rc0.11  Selettore modi operativi su MDI (semiautom)
)
ST   GESTCH3.xHold                * comando Hold al canale (esterno)

LD   GESTCH0.xEmer
ST   GESTCH3.xEmer                * comando Emergenza al canale (esterno)

LD   3333
ST   GESTCH3.xPPNumber            * numero part program da eseguire

LD   ALWAYS_ONE                    ** PLCFLAGS.1  Flag sempre stato on
ST   GESTCH3.xDisBlkSrc             * Disable channel block search

LD   %PLCFLAGS.0
ST   GESTCH3.xBlkSearch
ST   GESTCH3.xIntBlkSrc    * Forzam. esec. ricerca blocco interna
ST   GESTCH3.xOverstore  * Ab. overstore dopo ricerca blocco (provv.)

LD   ChannelFeedrate               ** feedrate for channel
ST   GESTCH3.xOverride

CAL  GESTCH3

LD   PulsAuxComand                 ** (gPlc2.28)Comando abilitazione da pulsantiera ausiliaria
JMPCN OVRTRE
LD   %cn0.rc2
ST   %cn3.rc2
OVRTRE:

LD   GESTCH3.yProgramRun * Programma in corso
ST   PRGRUN_CN3                    ** M0.2 cn3.rc8.0  Programma in corso

LD   BCO_STB_GET                   ** rc8.17 Strobe per GET resources
AND  AxStopSincGRP                 ** (gPlc13.11)Assi Fermi per sincronismo GRP[ax]
ST   BCI_ACK_GET                   ** rc0.29  ACK per GET resource

**************************
* FUNZIONI M CANALE 3 ****
**************************

* FUNZIONI M PER SINCRINISMI CON CANALE PRINCIPALE PER LA GESTIONE DELLA G800 E G 840*

LD   %rc9                * Registro funzioni M canale 0  (mauro)
EQ   30000
AND  %rc8.4              * Strobe funzioni M canale 0
ST   M30000_CN3                    ** M0.5 M30000_CN3: Attendi Servizio per Unit_1[(M10000 iniziolav.) / M10001(finelav.)]

LD   %rc9                * Registro funzioni M canale 0
EQ   30010
AND  %rc8.4              * Strobe funzioni M canale 0
ST   M30010_CN3                    ** M0.6 Sblocco Richiesta servizio (M10000_CN0 inizialavorazione)

LD   %rc9                * Registro funzioni M canale 0
EQ   30011
AND  %rc8.4              * Strobe funzioni M canale 0
ST   M30011_CN3                    ** M0.7 Sblocco Richiesta servizio (M10001_CN0 finelavorazione)

*******************************************************************************
*   HEAD1: X axis (30)
*******************************************************************************
PATH %ax30
PATH %ax_lsref30

***************************************
*   POWER ON (PON)
***************************************
LD   %pa3.31            * Simulato
*OR(
*LDN  %cn3.cc1.3           * Maschera assi associata al canale 0 U
*ANDN %cn3.cc1.4           * Maschera assi associata al canale 0 V
*)
ORN  %cn3.cc1.0
OR(
LD   %nvel11            ** 1=Mechatrolink
EQ   1
AND  %ring.drv4.RDD_wStatus.4 * PON
)
OR(
LD   %nvel11            ** 3,4=CANopen, Ecat
EQ   3
)
OR(
LD   %nvel11            ** 3,4=CANopen, Ecat
EQ   4
)
OR  (
LD   I_I_READY_DRIVE_UV            ** Ready signal drive U/V
AND  (
LD   %ax30.nvel11
EQ   0
)
)
ST   Pon_ax30                      ** PON Axe U (30)
***************************************

LDN  %cn3.cc1.0           * Maschera assi associata al canale 0
JMPC no_u_real

LD   %lsrefmode
ST   AXLSREF30.x_REF_mode        * 0=use ref switch...

LD   %lsreflevel
ST   AXLSREF30.x_TYPE_LS         * (1=NC, 0=NO)

LD   I_I_FC_UV_NEG                 ** U/V minimumm limit switch
ST   AXLSREF30.x_MIN_LS          * Min Limit switch

LD   I_I_FC_UV_POS                 ** Z1 maximun limit switch
ST   AXLSREF30.x_MAX_LS          * Max Limit switch

LD   I_I_INDEX_UV1                 ** U/V1 Axis Homing Switch
ST   AXLSREF30.x_REF_S           * Reference switch

CAL  AXLSREF30

LD   AXLSREF30.y_MIN_LS          * Min Limit switch
ST   GESTAX30.xMinusLS           * Negative limit switch

LD   AXLSREF30.y_MAX_LS          * Max Limit switch
ST   GESTAX30.xPlusLS            * Positive limit switch

LD   AXLSREF30.y_REF_S           * Reference switch
ST   GESTAX30.xRefLS             * Reference

LD   TON_ABIL.Q          * Abilitazione drives
ANDN TOF_MALARM.Q        * Assi in allarme
AND  Pon                           ** PON
ST   GESTAX30.xCloseLoop

LD   GSTMAC.yChSelMask.3
AND  SEL_ASSE.yExtMask.0
ANDN GESTAX9.xSelected              * Asse Lente selezionato
ANDN BUP_JOGOPEN                   ** ui16.16 Selezione esecuzione JOG a loop aperto
ST   GESTAX30.xSelected

***************************************
* Change REF quota for ABS reference
***************************************
CAL  RTRIG_AX_SEL30(CLK:=GESTAX30.xSelected)
LD   RTRIG_AX_SEL30.Q
JMPCN NoSel30
LD   ActualQtaAbsRef               ** Absolute homing quota
ST   QtaRefAbsSet                  ** Absolute homing quota setting
NoSel30:

LD   GESTAX30.xSelected
AND  %nvel14.0                     * Se Vale 1 ?gestito "Encoder Assoluto" (Da Configura Asse)
AND (
LD   ActualQtaAbsRef               ** Absolute homing quota
NE   QtaRefAbsSet                  ** Absolute homing quota setting
)
JMPCN NoEq30

LD   QtaRefAbsSet                  ** Absolute homing quota setting
ST   ActualQtaAbsRef               ** Absolute homing quota
NoEq30:
***************************************

LD   JOY_U_P                       **(gPlc2.7)Joystik U + selezionato
OR   (
LD   Pul_Jogp                      ** (gPlc0.4)jog+ pushbutton
AND  GESTAX30.xSelected
)
AND  EnabJogRTCP                   ** Abilita Jog RTCP
ANDN EMER_GEN                      ** M0.10 Emergenza generale
AND  GESTAX30.xCloseLoop
ST   GESTAX30.xJogPlus
R    %PLCmsg8.5

LD   JOY_U_M					   **(gPlc2.8)Joystik U - selezionato
OR   (
LD   Pul_Jogm                      ** (gPlc0.5)jog- pushbutton
AND  GESTAX30.xSelected
)
AND  EnabJogRTCP                   ** Abilita Jog RTCP
ANDN EMER_GEN                      ** M0.10 Emergenza generale
ANDN(
LD   %PLCerr20.20
AND   Pul_Jogp
)
AND  GESTAX30.xCloseLoop
ST   GESTAX30.xJogMinus

LD   BlcAvX1_user                  ** M74.0 Blocco avanzamento asse X1 da user.plc
OR   HoldSafePipeX                 ** (LsPlc26.2) Hold moving for X axis, not allow manual movement in pipe area
OR   MOVE_AXIS30.yHoldMov
OR   (
LD   AncolliXW_yHoldMov
OR   CMD_HOLDMOVING_CH3.0          ** M202 Hold moving command axis CH3 (bit0=X, bit1=Y...)
ANDN GESTAX30.xJogPlus
ANDN ch0_in_ref                    ** channel 0 in ref
)
ST   GESTAX30.xHoldMoving          * Richiesta blocco avanzamento

LD   MOVE_AXIS30.yFromPlc
OR   UsrGrantPlcMoveX
ST   GESTAX30.xFromPlc

LD   Res_Axes                      ** (gPlc25.1) reset axes disable electric shaft
ST   GESTAX30.xUnlock

LD   %nvel14.0                     * Se Vale 1 ?gestito "Encoder Assoluto" (Da Configura Asse)
ST   GESTAX30.xZeroForced          * Forzamento asse tarato

LDN  ch3_in_ref                    ** channel 3 in ref
ANDN EnJogRtcp                     ** (gPlc0.18)Abilitazione Jog RTCP tuning
*ANDN LimitSpeed
ST   GESTAX30.xEnFIR               * Abilita filtri FIR
ST   GESTAX30.xEnFrComp            ** Abilita friction compensation

LD   ALWAYS_ZERO                   ** PLCFLAGS.0  Flag sempre stato off
ST   GESTAX30.xDisLimiter

LD   %cn0.rc8.3            * ch0 in alarm
OR   %cn3.rc8.3            * ch3 in alarm
OR   EmerINC
ST   GESTAX30.xSetAlarm     ** Forzamento allarme asse

CAL  GESTAX30

LD   JOGrunning                    ** One axis moving in JOG
OR   %ra19.1         * Stato JOG all'interno del canale
ST   JOGrunning                    ** One axis moving in JOG

LD   REFrunning                    ** One axis moving in REF
OR   %ra19.2
ST   REFrunning                    ** One axis moving in REF

LD   INCrunning                    ** One axis moving in INC
OR   %ra19.3
ST   INCrunning                    ** One axis moving in INC

LD   GESTAX30.yDriveNotEn
S    %PLCerr2.3                    * Axis 30, drive not enable

no_u_real:

*******************************************************************************
*   HEAD1: Y (28) axis
*******************************************************************************
PATH %ax28
PATH %ax_lsref28

***************************************
*   POWER ON (PON)
***************************************
LD   %pa3.31            * Simulato
ORN  %cn3.cc1.1           * Maschera assi associata al canale 3 Y
OR(
LD   %nvel11            ** 1=Mechatrolink
EQ   1
AND  %ring.drv2.RDD_wStatus.4 * PON
)
OR(
LD   %nvel11            ** 3,4=CANopen, Ecat
EQ   3
)
OR(
LD   %nvel11            ** 3,4=CANopen, Ecat
EQ   4
)
OR  (
LD   I_I_READY_DRIVE_Y             ** Ready signal drive Y
AND  (
LD   %ax28.nvel11
EQ   0
)
)
ST   Pon_YT1                       ** PON Axe Y_T1
***************************************

LD  %cn3.cc1.1           * Maschera assi associata al canale 0
JMPCN NOAX28

LD   %lsrefmode
ST   AXLSREF28.x_REF_mode        * 0=use ref switch...

LD   %lsreflevel
ST   AXLSREF28.x_TYPE_LS         * (1=NC, 0=NO)

LD   I_I_FC_Y1_NEG                 ** Y1 minimumm limit switch
ST   AXLSREF28.x_MIN_LS          * Min Limit switch

LD   I_I_FC_Y1_POS                 ** Y1 maximun limit switch
ST   AXLSREF28.x_MAX_LS          * Max Limit switch

LD   I_I_INDEX_Y1                  ** Y1 Axis Homing Switch
ST   AXLSREF28.x_REF_S           * Reference switch

CAL  AXLSREF28

LD   AXLSREF28.y_MIN_LS          * Min Limit switch
ST   GESTAX28.xMinusLS           * Negative limit switch

LD   AXLSREF28.y_MAX_LS          * Max Limit switch
ST   GESTAX28.xPlusLS            * Positive limit switch

LD   AXLSREF28.y_REF_S           * Reference switch
ST   GESTAX28.xRefLS             * Reference

LD   TON_ABIL.Q                  * Abilitazione drives
ANDN TOF_MALARM.Q                * Assi in allarme
AND  Pon                           ** PON
ST   GESTAX28.xCloseLoop

LD   GSTMAC.yChSelMask.3
AND  SEL_ASSE.yExtMask.1
ANDN PulsAuxComand                 ** (gPlc2.28)Comando abilitazione da pulsantiera ausiliaria
OR   I_HW_Y_SEL_USR                ** (gPlc2.24)Y selected da volantino pulsantiera ausiliaria
OR   Gui_Pul_Y_M
OR   Gui_Pul_Y_P
ANDN GESTAX9.xSelected              * Asse Lente selezionato
ANDN BUP_JOGOPEN                   ** ui16.16 Selezione esecuzione JOG a loop aperto
ST   GESTAX28.xSelected

***************************************
* Change REF quota for ABS reference
***************************************
CAL  RTRIG_AX_SEL28(CLK:=GESTAX28.xSelected)
LD   RTRIG_AX_SEL28.Q
JMPCN NoSel28
LD   ActualQtaAbsRef               ** Absolute homing quota
ST   QtaRefAbsSet                  ** Absolute homing quota setting
NoSel28:

LD   GESTAX28.xSelected
AND  %nvel14.0                     * Se Vale 1 ?gestito "Encoder Assoluto" (Da Configura Asse)
AND (
LD   ActualQtaAbsRef               ** Absolute homing quota
NE   QtaRefAbsSet                  ** Absolute homing quota setting
)
JMPCN NoEq28

LD   QtaRefAbsSet                  ** Absolute homing quota setting
ST   ActualQtaAbsRef               ** Absolute homing quota
NoEq28:
***************************************

LD   JOY_Y_P                       ** (gPlc0.16)Joystik Y + selezionato
OR   Gui_Pul_Y_P
OR (
LD   Pul_Jogp                      ** (gPlc0.4)jog+ pushbutton
AND  GESTAX28.xSelected
)
AND  EnabJogRTCP                   ** Abilita Jog RTCP
ANDN EMER_GEN                      ** M0.10 Emergenza generale
AND  GESTAX28.xCloseLoop
ST   GESTAX28.xJogPlus

LD   GESTAX28.xJogPlus
OR   (
LD   GSTMAC.xPlus
AND  GESTAX28.xSelected
)
ST   OrderMoveYPosit               ** (LsPlc26.5) Order of movement positive dir for Y

LD   JOY_Y_M                       ** (gPlc0.17)Joystik Y - selezionato
OR   Gui_Pul_Y_M
OR (
LD   Pul_Jogm                      ** (gPlc0.5)jog- pushbutton
AND  GESTAX28.xSelected
)
AND  EnabJogRTCP                   ** Abilita Jog RTCP
ANDN EMER_GEN                      ** M0.10 Emergenza generale
AND  GESTAX28.xCloseLoop
ST   GESTAX28.xJogMinus

LD   GESTAX28.xJogMinus
OR   (
LD   GSTMAC.xMinus
AND  GESTAX28.xSelected
)
ST   OrderMoveYNegat               ** (LsPlc26.6) Order of movement negative dir for Y

LD   %nvel14.0                     * Se Vale 1 ?gestito "Encoder Assoluto" (Da Configura Asse)
ST   GESTAX28.xZeroForced * Forzamento asse tarato

LD   GESTAX1.xHoldMoving           * Richiesta blocco avanzamento
OR   BlcAvY1_user                  ** M74.4 Blocco avanzamento asse Y da user.plc
OR   HoldSafePipeY                 ** (LsPlc26.7) Hold moving for Y axis, not allow manual movement in pipe area
OR   CMD_HOLDMOVING_CH3.1          ** M202 Hold moving command axis CH3 (bit0=X, bit1=Y...)
ST   GESTAX28.xHoldMoving          * Richiesta blocco avanzamento

LD   Res_Axes                      ** (gPlc25.1) reset axes disable electric shaft
ST   GESTAX28.xUnlock

LDN  ch3_in_ref                    ** channel 3 in ref
ANDN EnJogRtcp                     ** (gPlc0.18)Abilitazione Jog RTCP tuning
ST   GESTAX28.xEnFIR               * Abilita filtri FIR
ST   GESTAX28.xEnFrComp            ** Abilita friction compensation

LD   ALWAYS_ZERO                   ** PLCFLAGS.0  Flag sempre stato off
ST   GESTAX28.xDisLimiter

LD   %cn0.rc8.3            * ch0 in alarm
OR   %cn3.rc8.3            * ch3 in alarm
OR   EmerINC
ST   GESTAX28.xSetAlarm     ** Forzamento allarme asse

CAL  GESTAX28

LD   JOGrunning                    ** One axis moving in JOG
OR   %ra19.1         * Stato JOG all'interno del canale
ST   JOGrunning                    ** One axis moving in JOG

LD   REFrunning                    ** One axis moving in REF
OR   %ra19.2
ST   REFrunning                    ** One axis moving in REF

LD   INCrunning                    ** One axis moving in INC
OR   %ra19.3
ST   INCrunning                    ** One axis moving in INC

LD   GESTAX28.yDriveNotEn
S    %PLCerr2.1                    * Axis 28, drive not enable

LD   %pa9                * Velocit?massima asse
MUL  1000
DIV  60
ST   %ra50               * Limitazione velocita' massima interpolazione

LD   BSG_INC                       ** rg1.2 Selezione modo INC (inc.fissi)
JMPCN SVIX28

LD   %pa59               * Velocit?di Repos
MUL  1000
DIV  60
MUL  AxesOverride                  ** (gPlc16) feed degli assi (%)
DIV  100
ST   %ra50               * Limitazione velocita' massima interpolazione

SVIX28:
NOAX28:

*******************************************************************************
*   HEAD1: Z (29) axis
*******************************************************************************
PATH %ax29
PATH %ax_lsref29

***************************************
*   POWER ON (PON)
***************************************
LD   %pa3.31            * Simulato
ORN  %cn3.cc1.2         * Maschera assi associata al canale
OR(
LD   %nvel11            ** 1=Mechatrolink
EQ   1
AND  %ring.drv3.RDD_wStatus.4 * PON
)
OR(
LD   %nvel11            ** 3,4=CANopen, Ecat
EQ   3
)
OR(
LD   %nvel11            ** 3,4=CANopen, Ecat
EQ   4
)
OR  (
LD   I_I_READY_DRIVE_Z             ** Ready signal drive Z
AND  (
LD   %ax29.nvel11
EQ   0
)
)
ST   Pon_ZT1                       ** PON Axe Y_T1
***************************************

LD  %cn3.cc1.2           * Maschera assi associata al canale 0
JMPCN NOAX29

LD   %lsrefmode
ST   AXLSREF29.x_REF_mode        * 0=use ref switch...

LD   %lsreflevel
ST   AXLSREF29.x_TYPE_LS         * (1=NC, 0=NO)

LD   I_I_FC_Z1_NEG                 ** Z1 minimumm limit switch
ST   AXLSREF29.x_MIN_LS          * Min Limit switch

LD   I_I_FC_Z1_POS                 ** Z1 maximun limit switch
ST   AXLSREF29.x_MAX_LS          * Max Limit switch

LD   I_I_INDEX_Z1                  ** Z1 Axis Homing Switch
ST   AXLSREF29.x_REF_S           * Reference switch

CAL  AXLSREF29

LD   AXLSREF29.y_MIN_LS          * Min Limit switch
ST   GESTAX29.xMinusLS           * Negative limit switch

LD   AXLSREF29.y_MAX_LS          * Max Limit switch
ST   GESTAX29.xPlusLS            * Positive limit switch

LD   AXLSREF29.y_REF_S           * Reference switch
ST   GESTAX29.xRefLS             * Reference

LD   TON_ABIL.Q                     * Abilitazione drives
ANDN TOF_MALARM.Q                   * Assi in allarme
AND  Pon                           ** PON
ST   GESTAX29.xCloseLoop

LD   GSTMAC.yChSelMask.3
AND  SEL_ASSE.yExtMask.2
ANDN PulsAuxComand                 ** (gPlc2.28)Comando abilitazione da pulsantiera ausiliaria
OR   I_HW_Z_SEL_USR                ** (gPlc2.25)Z selected da volantino pulsantiera ausiliaria
OR   Gui_Pul_Z_M
OR   Gui_Pul_Z_P
ANDN GESTAX9.xSelected              * Asse Lente selezionato
ANDN BUP_JOGOPEN                   ** ui16.16 Selezione esecuzione JOG a loop aperto
ST   GESTAX29.xSelected

***************************************
* Change REF quota for ABS reference
***************************************
CAL  RTRIG_AX_SEL29(CLK:=GESTAX29.xSelected)
LD   RTRIG_AX_SEL29.Q
JMPCN NoSel29
LD   ActualQtaAbsRef               ** Absolute homing quota
ST   QtaRefAbsSet                  ** Absolute homing quota setting
NoSel29:

LD   GESTAX29.xSelected
AND  %nvel14.0                     * Se Vale 1 ?gestito "Encoder Assoluto" (Da Configura Asse)
AND (
LD   ActualQtaAbsRef               ** Absolute homing quota
NE   QtaRefAbsSet                  ** Absolute homing quota setting
)
JMPCN NoEq29

LD   QtaRefAbsSet                  ** Absolute homing quota setting
ST   ActualQtaAbsRef               ** Absolute homing quota
NoEq29:
***************************************

LD   JOY_Z_P					   **(gPlc19.3)Joystik Z + selezionato
OR   Gui_Pul_Z_P
OR   (
LD   Pul_Jogp                      ** (gPlc0.4)jog+ pushbutton
AND  GESTAX29.xSelected
)
OR   I_I_PUL_TORCH_UP              ** Jog+ pushbutton (Torch Up)
AND(
LD   ch0_in_aut                    ** channel 0 in aut
OR   ch3_in_jog                    ** channel 3 in jog
OR   ch3_in_inc                    ** channel 3 in inc
)
AND  EnabJogRTCP                   ** Abilita Jog RTCP
ANDN EMER_GEN                      ** M0.10 Emergenza generale
AND  GESTAX29.xCloseLoop
ST   GESTAX29.xJogPlus

LD   JOY_Z_M                       **(gPlc19.4)Joystik Z - selezionato
OR   Gui_Pul_Z_M
OR   (
LD   Pul_Jogm                      ** (gPlc0.5)jog- pushbutton
AND  GESTAX29.xSelected
)
OR   I_I_PUL_TORCH_DW              ** Jog- pushbutton (Torch Down)
AND(
LD   ch3_in_aut                    ** channel 3 in aut
OR   ch3_in_jog                    ** channel 3 in jog
OR   ch3_in_inc                    ** channel 3 in inc
)
AND  EnabJogRTCP                   ** Abilita Jog RTCP
ANDN EMER_GEN                      ** M0.10 Emergenza generale
AND  GESTAX29.xCloseLoop
ST   GESTAX29.xJogMinus

LD   ALWAYS_ONE                    ** PLCFLAGS.1  Flag sempre stato on
ST   GESTAX29.xBrakeEnab

LD   CS_X_Overtravel               ** (gPlc13.12)Camma sw asse X oltre limite max
OR   (
  LD      %PLCerr5.4      **PLC Err 164 Tip touch (A11=1, A14=0, A15=0 in normal operation)
  ANDN Pul_Jogp                      ** (gPlc0.4)jog+ pushbutton
)
OR   CMD_HOLDMOVING_CH3.2           ** M202 Hold moving command axis CH3 (bit0=X, bit1=Y...)
ST   GESTAX29.xHoldMoving * Richiesta blocco avanzamento

LD   %nvel14.0                     * Se Vale 1 ?gestito "Encoder Assoluto" (Da Configura Asse)
ST   GESTAX29.xZeroForced * Forzamento asse tarato

LDN  ch3_in_ref                    ** channel 3 in ref
ANDN EnJogRtcp                     ** (gPlc0.18)Abilitazione Jog RTCP tuning
ANDN DisabFir_CH3_axes.2
ST   GESTAX29.xEnFIR               * Abilita filtri FIR
ST   GESTAX29.xEnFrComp            ** Abilita friction compensation

LD   ALWAYS_ZERO                   ** PLCFLAGS.0  Flag sempre stato off
ST   GESTAX29.xDisLimiter

LD   Res_Axes                      ** (gPlc25.1) reset axes disable electric shaft
ST   GESTAX29.xUnlock

LD   %cn0.rc8.3            * ch0 in alarm
OR   %cn3.rc8.3            * ch3 in alarm
OR   EmerINC
ST   GESTAX29.xSetAlarm     ** Forzamento allarme asse

CAL  GESTAX29

LD   JOGrunning                    ** One axis moving in JOG
OR   %ra19.1         * Stato JOG all'interno del canale
ST   JOGrunning                    ** One axis moving in JOG

LD   REFrunning                    ** One axis moving in REF
OR   %ra19.2
ST   REFrunning                    ** One axis moving in REF

LD   INCrunning                    ** One axis moving in INC
OR   %ra19.3
ST   INCrunning                    ** One axis moving in INC

LD   GESTAX29.yDriveNotEn
S    %PLCerr2.2                    * Axis 29, drive not enable

LD   %vrtc5.VrdwCtrlRegister0.18 * De overlap
JMPCN NOAX29DeOverlap

LD   0
ST   %ra50               * Limitazione velocita' massima interpolazione

NOAX29DeOverlap:

LD   GESTAX29.yBrake
ST   O_O_BRAKE_Z1                  ** Brake Z1 axis

NOAX29:
*******************************************************************************
*   HEAD1: U (27) axis
*******************************************************************************
PATH %ax27
PATH %ax_lsref27

***************************************
*   POWER ON (PON)
***************************************
LD   %pa3.31            * Simulato
ORN  %cn3.cc1.3         * Maschera assi associata al canale
OR(
LD   %nvel11            ** 1=Mechatrolink
EQ   1
AND  %ring.drv1.RDD_wStatus.4 * PON
)
OR(
LD   %nvel11            ** 3,4=CANopen, Ecat
EQ   3
)
OR(
LD   %nvel11            ** 3,4=CANopen, Ecat
EQ   4
)
OR  (
LD   I_I_READY_DRIVE_X             ** Ready signal drive X
AND  (
LD   %ax27.nvel11
EQ   0
)
)
ST   Pon_XT1                       ** PON Axe X_T1
***************************************

LD  %cn3.cc1.3           * Maschera assi associata al canale 0
JMPCN NOAX27

***
*   LIMIT SWITCH & REFERENCE SWITCH

LD   %lsrefmode
ST   AXLSREF27.x_REF_mode        * 0=use ref switch...

LD   %lsreflevel
ST   AXLSREF27.x_TYPE_LS         * (1=NC, 0=NO)

LD   I_I_FC_X1_NEG                 ** X1 minimumm limit switch
ST   AXLSREF27.x_MIN_LS          * Min Limit switch

LD   I_I_FC_X1_POS                 ** X1 maximun limit switch
ST   AXLSREF27.x_MAX_LS          * Max Limit switch

LD   I_I_INDEX_X1                  ** X1 Axis Homing Switch
ST   AXLSREF27.x_REF_S           * Reference switch

CAL  AXLSREF27

LD   AXLSREF27.y_MIN_LS          * Min Limit switch
ST   GESTAX27.xMinusLS           * Negative limit switch

LD   AXLSREF27.y_MAX_LS          * Max Limit switch
ST   GESTAX27.xPlusLS            * Positive limit switch

LD   AXLSREF27.y_REF_S           * Reference switch
ST   GESTAX27.xRefLS             * Reference
***

LD   TON_ABIL.Q          * Abilitazione drives
ANDN TOF_MALARM.Q        * Assi in allarme
AND  Pon                           ** PON
ST   GESTAX27.xCloseLoop

LD   GSTMAC.yChSelMask.3
AND  SEL_ASSE.yExtMask.3
ANDN PulsAuxComand                 ** (gPlc2.28)Comando abilitazione da pulsantiera ausiliaria
OR   I_HW_X_SEL_USR                ** (gPlc2.23)X selected da volantino pulsantiera ausiliaria
ANDN GESTAX9.xSelected              * Asse Lente selezionato
ANDN BUP_JOGOPEN                   ** ui16.16 Selezione esecuzione JOG a loop aperto
AND  ALWAYS_ZERO
ST   GESTAX27.xSelected

***************************************
* Change REF quota for ABS reference
***************************************
CAL  RTRIG_AX_SEL27(CLK:=GESTAX27.xSelected)
LD   RTRIG_AX_SEL27.Q
JMPCN NoSel27
LD   ActualQtaAbsRef               ** Absolute homing quota
ST   QtaRefAbsSet                  ** Absolute homing quota setting
NoSel27:

LD   GESTAX27.xSelected
AND  %nvel14.0                     * Se Vale 1 ?gestito "Encoder Assoluto" (Da Configura Asse)
AND (
LD   ActualQtaAbsRef               ** Absolute homing quota
NE   QtaRefAbsSet                  ** Absolute homing quota setting
)
JMPCN NoEq27

LD   QtaRefAbsSet                  ** Absolute homing quota setting
ST   ActualQtaAbsRef               ** Absolute homing quota
NoEq27:
***************************************

LD   JOY_X_P                       ** (gPlc0.14)Joystik X + selezionato
OR (
LD   Pul_Jogp                      ** (gPlc0.4)jog+ pushbutton
AND  GESTAX27.xSelected
)
AND  EnabJogRTCP                   ** Abilita Jog RTCP
ANDN EMER_GEN                      ** M0.10 Emergenza generale
AND  GESTAX27.xCloseLoop
ST   GESTAX27.xJogPlus

LD   GESTAX27.xJogPlus
OR   (
LD   GSTMAC.xPlus
AND  GESTAX27.xSelected
)
ST   OrderMoveXPosit               ** (LsPlc26.3) Order of movement positive dir for X

LD   JOY_X_M                       ** (gPlc0.15)Joystik X - selezionato
OR (
LD   Pul_Jogm                      ** (gPlc0.5)jog- pushbutton
AND  GESTAX27.xSelected
)
AND  EnabJogRTCP                   ** Abilita Jog RTCP
ANDN EMER_GEN                      ** M0.10 Emergenza generale
AND  GESTAX27.xCloseLoop
ST   GESTAX27.xJogMinus

LD   GESTAX27.xJogMinus
OR   (
LD   GSTMAC.xMinus
AND  GESTAX27.xSelected
)
ST   OrderMoveXNegat               ** (LsPlc26.4) Order of movement negative dir for X

LD   %nvel14.0                     * Se Vale 1 ?gestito "Encoder Assoluto" (Da Configura Asse)
ST   GESTAX27.xZeroForced          * Forzamento asse tarato

LD   GESTAX0.xHoldMoving           * Richiesta blocco avanzamento
OR   BlcAvX1_user                  ** M74.0 Blocco avanzamento asse X1 da user.plc
OR   HoldSafePipeX                 ** (LsPlc26.2) Hold moving for X axis, not allow manual movement in pipe area
OR   CMD_HOLDMOVING_CH3.0          ** M202 Hold moving command axis CH3 (bit0=X, bit1=Y...)
ST   GESTAX27.xHoldMoving          * Richiesta blocco avanzamento

LD   Res_Axes                      ** (gPlc25.1) reset axes disable electric shaft
ST   GESTAX27.xUnlock

LDN  ch3_in_ref                    ** channel 3 in ref
ANDN EnJogRtcp                     ** (gPlc0.18)Abilitazione Jog RTCP tuning
ST   GESTAX27.xEnFIR               * Abilita filtri FIR
ST   GESTAX27.xEnFrComp            ** Abilita friction compensation

LD   ALWAYS_ZERO                   ** PLCFLAGS.0  Flag sempre stato off
ST   GESTAX27.xDisLimiter

LD   %cn0.rc8.3            * ch0 in alarm
OR   %cn3.rc8.3            * ch3 in alarm
OR   EmerINC
ST   GESTAX27.xSetAlarm     ** Forzamento allarme asse

CAL  GESTAX27

LD   JOGrunning                    ** One axis moving in JOG
OR   %ra19.1         * Stato JOG all'interno del canale
ST   JOGrunning                    ** One axis moving in JOG

LD   REFrunning                    ** One axis moving in REF
OR   %ra19.2
ST   REFrunning                    ** One axis moving in REF

LD   INCrunning                    ** One axis moving in INC
OR   %ra19.3
ST   INCrunning                    ** One axis moving in INC

LD   GESTAX27.yDriveNotEn
S    %PLCerr2.0                    * Axis 27, drive not enable

LD   %pa9                * Velocit?massima asse
MUL  1000
DIV  60
ST   %ra50               * Limitazione velocita' massima interpolazione

LD   BSG_INC                       ** rg1.2 Selezione modo INC (inc.fissi)
JMPCN SVIX27

LD   %pa59               * Velocit?di Repos
MUL  1000
DIV  60
MUL  AxesOverride                  ** (gPlc16) feed degli assi (%)
DIV  100
ST   %ra50               * Limitazione velocita' massima interpolazione

SVIX27:
NOAX27:

*******************************************************************************
*   HEAD1: V axis (31) slave spindle axis
*******************************************************************************
PATH %ax31
PATH %ax_lsref31

***************************************
*   POWER ON (PON)
***************************************
LD   %pa3.31            * Simulato
OR(
LD   %nvel11            ** 1=Mechatrolink
EQ   1
AND  %ring.drv4.RDD_wStatus.4 * PON
)
OR(
LD   %nvel11            ** 3,4=CANopen, Ecat
EQ   3
)
OR(
LD   %nvel11            ** 3,4=CANopen, Ecat
EQ   4
)
OR  (
LD   I_I_READY_DRIVE_UV            ** Ready signal drive U/V
AND  (
LD   %ax30.nvel11
EQ   0
)
)
ST   Pon_ax31                      ** PON Axe U (30)
***************************************

LDN  %cn3.cc1.4           * Maschera assi associata al canale 0
JMPC no_v_real

LD   %lsrefmode
ST   AXLSREF31.x_REF_mode        * 0=use ref switch...

LD   %lsreflevel
ST   AXLSREF31.x_TYPE_LS         * (1=NC, 0=NO)

LD   I_I_FC_V_NEG                 ** U/V minimumm limit switch
ST   AXLSREF31.x_MIN_LS          * Min Limit switch

LD   I_I_FC_V_POS                 ** Z1 maximun limit switch
ST   AXLSREF31.x_MAX_LS          * Max Limit switch

LD   I_I_INDEX_V                 ** U/V1 Axis Homing Switch
ST   AXLSREF31.x_REF_S           * Reference switch

CAL  AXLSREF31

LD   AXLSREF31.y_MIN_LS          * Min Limit switch
ST   GESTAX31.xMinusLS           * Negative limit switch

LD   AXLSREF31.y_MAX_LS          * Max Limit switch
ST   GESTAX31.xPlusLS            * Positive limit switch

LD   AXLSREF31.y_REF_S           * Reference switch
ST   GESTAX31.xRefLS             * Reference

LD   TON_ABIL.Q          * Abilitazione drives
ANDN TOF_MALARM.Q        * Assi in allarme
AND  Pon                           ** PON
ST   GESTAX31.xCloseLoop

LD   GSTMAC.yChSelMask.3
AND  SEL_ASSE.yExtMask.4
OR(
LD   RemContrUPlus
AND  Rem_Combination
)
OR(
LD   RemContrUMinus
AND  Rem_Combination
)
OR   Gui_Pul_X1_M
OR   Gui_Pul_X1_P
ANDN GESTAX9.xSelected              * Asse Lente selezionato
ANDN BUP_JOGOPEN                   ** ui16.16 Selezione esecuzione JOG a loop aperto
ST   GESTAX31.xSelected

***************************************
* Change REF quota for ABS reference
***************************************
CAL  RTRIG_AX_SEL31(CLK:=GESTAX31.xSelected)
LD   RTRIG_AX_SEL31.Q
JMPCN NoSel31
LD   ActualQtaAbsRef               ** Absolute homing quota
ST   QtaRefAbsSet                  ** Absolute homing quota setting
NoSel31:

LD   GESTAX31.xSelected
AND  %nvel14.0                     * Se Vale 1 ?gestito "Encoder Assoluto" (Da Configura Asse)
AND (
LD   ActualQtaAbsRef               ** Absolute homing quota
NE   QtaRefAbsSet                  ** Absolute homing quota setting
)
JMPCN NoEq31

LD   QtaRefAbsSet                  ** Absolute homing quota setting
ST   ActualQtaAbsRef               ** Absolute homing quota
NoEq31:
***************************************

LD   Pul_Jogp                      ** (gPlc0.4)jog+ pushbutton
OR(
LD   RemContrUPlus
AND  Rem_Combination
)
OR   Gui_Pul_X1_P
AND  GESTAX31.xSelected
AND  EnabJogRTCP                   ** Abilita Jog RTCP
ANDN EMER_GEN                      ** M0.10 Emergenza generale
AND  GESTAX31.xSelected
AND  GESTAX31.xCloseLoop
ST   GESTAX31.xJogPlus

LD   Pul_Jogm                      ** (gPlc0.5)jog- pushbutton
OR(
LD   RemContrUMinus
AND  Rem_Combination
)
OR   Gui_Pul_X1_M
AND  GESTAX31.xSelected
AND  EnabJogRTCP                   ** Abilita Jog RTCP
ANDN EMER_GEN                      ** M0.10 Emergenza generale
AND  GESTAX31.xSelected
AND  GESTAX31.xCloseLoop
ST   GESTAX31.xJogMinus

LD   GESTAX6.xHoldMoving           * Richiesta blocco avanzamento
OR   BlcAvX1_user                  ** M74.0 Blocco avanzamento asse X1 da user.plc
OR   HoldSafePipeX                 ** (LsPlc26.2) Hold moving for X axis, not allow manual movement in pipe area
OR(
LD   CMD_HOLDMOVING_CH3.4          ** M202 Hold moving command axis CH3 (bit0=X, bit1=Y...)
ANDN GESTAX31.xJogMinus
ANDN ch0_in_ref                    ** channel 0 in ref
)
OR   (
LD   AncolliWV_yHoldMov
ANDN GESTAX31.xJogMinus
ANDN ch0_in_ref                    ** channel 0 in ref
)
ST   GESTAX31.xHoldMoving          * Richiesta blocco avanzamento

*LD   MOVE_AXIS31.yFromPlc
LD   UsrGrantPlcMoveX1
ST   GESTAX31.xFromPlc

LD   Res_Axes                      ** (gPlc25.1) reset axes disable electric shaft
ST   GESTAX31.xUnlock

LD   %nvel14.0                     * Se Vale 1 ?gestito "Encoder Assoluto" (Da Configura Asse)
ST   GESTAX31.xZeroForced          * Forzamento asse tarato

LDN  ch3_in_ref                    ** channel 3 in ref
ANDN EnJogRtcp                     ** (gPlc0.18)Abilitazione Jog RTCP tuning
ST   GESTAX31.xEnFIR               * Abilita filtri FIR
ST   GESTAX31.xEnFrComp            ** Abilita friction compensation

LD   ALWAYS_ZERO                   ** PLCFLAGS.0  Flag sempre stato off
ST   GESTAX31.xDisLimiter

LD   %cn0.rc8.3            * ch0 in alarm
OR   %cn3.rc8.3            * ch3 in alarm
OR   EmerINC
ST   GESTAX31.xSetAlarm     ** Forzamento allarme asse

CAL  GESTAX31

LD   JOGrunning                    ** One axis moving in JOG
OR   %ra19.1                       * Stato JOG all'interno del canale
ST   JOGrunning                    ** One axis moving in JOG

LD   REFrunning                    ** One axis moving in REF
OR   %ra19.2
ST   REFrunning                    ** One axis moving in REF

LD   INCrunning                    ** One axis moving in INC
OR   %ra19.3
ST   INCrunning                    ** One axis moving in INC

LD   GESTAX31.yDriveNotEn
S    %PLCerr2.15                    * Axis 30, drive not enable

no_v_real:

*******************************************************************************
*   HEAD1: w axis (36) slave spindle middle
*******************************************************************************
PATH %ax36
PATH %ax_lsref36

***************************************
*   POWER ON (PON)
***************************************
LD   %pa3.31            * Simulato
OR(
LD   %nvel11            ** 1=Mechatrolink
EQ   1
AND  %ring.drv4.RDD_wStatus.4 * PON
)
OR(
LD   %nvel11            ** 3,4=CANopen, Ecat
EQ   3
)
OR(
LD   %nvel11            ** 3,4=CANopen, Ecat
EQ   4
)
OR  (
LD   I_I_READY_DRIVE_UV            ** Ready signal drive U/V
AND  (
LD   %ax30.nvel11
EQ   0
)
)
ST   Pon_ax36                      ** PON Axe W (36)
***************************************

LDN  %cn3.cc1.5          * Maschera assi associata al canale 0
JMPC no_w_real

LD   %lsrefmode
ST   AXLSREF36.x_REF_mode        * 0=use ref switch...

LD   %lsreflevel
ST   AXLSREF36.x_TYPE_LS         * (1=NC, 0=NO)

LD   I_I_FC_W_NEG                 ** U/V minimumm limit switch
ST   AXLSREF36.x_MIN_LS          * Min Limit switch

LD   I_I_FC_W_POS                 ** Z1 maximun limit switch
ST   AXLSREF36.x_MAX_LS          * Max Limit switch

LD   I_I_INDEX_W                 ** U/V1 Axis Homing Switch
ST   AXLSREF36.x_REF_S           * Reference switch

CAL  AXLSREF36

LD   AXLSREF36.y_MIN_LS          * Min Limit switch
ST   GESTAX36.xMinusLS           * Negative limit switch

LD   AXLSREF36.y_MAX_LS          * Max Limit switch
ST   GESTAX36.xPlusLS            * Positive limit switch

LD   AXLSREF36.y_REF_S           * Reference switch
ST   GESTAX36.xRefLS             * Reference

LD   TON_ABIL.Q          * Abilitazione drives
ANDN TOF_MALARM.Q        * Assi in allarme
AND  Pon                           ** PON
ST   GESTAX36.xCloseLoop

LD   GSTMAC.yChSelMask.3
AND  SEL_ASSE.yExtMask.5
ANDN GESTAX9.xSelected              * Asse Lente selezionato
OR   Gui_Pul_X3_M
OR   Gui_Pul_X3_P
ANDN BUP_JOGOPEN                   ** ui16.16 Selezione esecuzione JOG a loop aperto
ST   GESTAX36.xSelected

***************************************
* Change REF quota for ABS reference
***************************************
CAL  RTRIG_AX_SEL36(CLK:=GESTAX36.xSelected)
LD   RTRIG_AX_SEL36.Q
JMPCN NoSel36
LD   ActualQtaAbsRef               ** Absolute homing quota
ST   QtaRefAbsSet                  ** Absolute homing quota setting
NoSel36:

LD   GESTAX36.xSelected
AND  %nvel14.0                     * Se Vale 1 ?gestito "Encoder Assoluto" (Da Configura Asse)
AND (
LD   ActualQtaAbsRef               ** Absolute homing quota
NE   QtaRefAbsSet                  ** Absolute homing quota setting
)
JMPCN NoEq36

LD   QtaRefAbsSet                  ** Absolute homing quota setting
ST   ActualQtaAbsRef               ** Absolute homing quota
NoEq36:
***************************************

LD   Pul_Jogp                      ** (gPlc0.4)jog+ pushbutton
AND  EnabJogRTCP                   ** Abilita Jog RTCP
OR   Gui_Pul_X3_P
ANDN EMER_GEN                      ** M0.10 Emergenza generale
AND  GESTAX36.xSelected
AND  GESTAX36.xCloseLoop
ST   GESTAX36.xJogPlus

LD   Pul_Jogm                      ** (gPlc0.5)jog- pushbutton
AND  EnabJogRTCP                   ** Abilita Jog RTCP
OR   Gui_Pul_X3_M
ANDN EMER_GEN                      ** M0.10 Emergenza generale
AND  GESTAX36.xSelected
AND  GESTAX36.xCloseLoop
ST   GESTAX36.xJogMinus

LD   GESTAX6.xHoldMoving           * Richiesta blocco avanzamento
OR   BlcAvX1_user                  ** M74.0 Blocco avanzamento asse X1 da user.plc
OR   HoldSafePipeX                 ** (LsPlc26.2) Hold moving for X axis, not allow manual movement in pipe area
OR(
     LD   Hold_moving_axW
     ANDN Gest5Ax
	 ANDN (
	      LD    %ra4
	      GE    0
	      AND   GESTAX36.xJogPlus
	 )
)
OR(
LD   AncolliWV_yHoldMov
OR   %PLCmsg8.9
ANDN GESTAX36.xJogPlus
)
OR(
LD   AncolliXW_yHoldMov
OR   %PLCmsg8.10
ANDN GESTAX36.xJogMinus
)
OR(
     LD   %ax71.ra24
     SUB  ParkingPositionUnload
     ABS
     GT   2000                        *[2mm]
	 AND(
	      LD   %ax36.ra24
		  LT   SafeDis_W_L1
	 )
     ANDN GESTAX36.xJogPlus
)
ANDN ch0_in_ref                    ** channel 0 in ref
ST   GESTAX36.xHoldMoving          * Richiesta blocco avanzamento
ST   GESTAX36_xHoldMoving

LD   Res_Axes                      ** (gPlc25.1) reset axes disable electric shaft
ST   GESTAX36.xUnlock

LD   %nvel14.0                     * Se Vale 1 ?gestito "Encoder Assoluto" (Da Configura Asse)
ST   GESTAX36.xZeroForced          * Forzamento asse tarato

LDN  ch3_in_ref                    ** channel 3 in ref
ANDN EnJogRtcp                     ** (gPlc0.18)Abilitazione Jog RTCP tuning
ST   GESTAX36.xEnFIR               * Abilita filtri FIR
ST   GESTAX36.xEnFrComp            ** Abilita friction compensation

LD   ALWAYS_ZERO                   ** PLCFLAGS.0  Flag sempre stato off
ST   GESTAX36.xDisLimiter

LD   %cn0.rc8.3            * ch0 in alarm
OR   %cn3.rc8.3            * ch3 in alarm
OR   EmerINC
ST   GESTAX36.xSetAlarm     ** Forzamento allarme asse

CAL  GESTAX36

LD   JOGrunning                    ** One axis moving in JOG
OR   %ra19.1                       * Stato JOG all'interno del canale
ST   JOGrunning                    ** One axis moving in JOG

LD   REFrunning                    ** One axis moving in REF
OR   %ra19.2
ST   REFrunning                    ** One axis moving in REF

LD   INCrunning                    ** One axis moving in INC
OR   %ra19.3
ST   INCrunning                    ** One axis moving in INC

LD   GESTAX36.yDriveNotEn
S    %PLCerr2.19                    * Axis 30, drive not enable

no_w_real:

*******************************************************************************
*   HEAD1: A (32) axis
*******************************************************************************
PATH %ax32
PATH %ax_lsref32

***************************************
*   POWER ON (PON)
***************************************
LD   %pa3.31            * Simulato
ORN  %cn3.cc1.6         * Maschera assi associata al canale
OR(
LD   %nvel11            ** 1=Mechatrolink
EQ   1
AND  %ring.drv1.RDD_wStatus.4 * PON
)
OR(
LD   %nvel11            ** 3,4=CANopen, Ecat
EQ   3
)
OR(
LD   %nvel11            ** 3,4=CANopen, Ecat
EQ   4
)
OR   (
LD   I_I_READY_DRIVE_A             ** Ready signal drive A
AND  (
LD   %ax9.nvel11
EQ   0
)
)
ST   Pon_A                         ** PON Axe A

LD  %cn3.cc1.6           * Maschera assi associata al canale 0
JMPCN NOAX32

***
*   LIMIT SWITCH & REFERENCE SWITCH

LD   %lsrefmode
ST   AXLSREF32.x_REF_mode        * 0=use ref switch...

LD   %lsreflevel
ST   AXLSREF32.x_TYPE_LS         * (1=NC, 0=NO)

LD   I_I_FC_A1_NEG                 ** A1 minimumm limit switch
ST   AXLSREF32.x_MIN_LS          * Min Limit switch

LD   I_I_FC_A1_POS                 ** A1 maximun limit switch
ST   AXLSREF32.x_MAX_LS          * Max Limit switch

LD   I_I_INDEX_A1                  ** A1 Axis Homing Switch
ST   AXLSREF32.x_REF_S           * Reference switch

CAL  AXLSREF32

LD   AXLSREF32.y_MIN_LS          * Min Limit switch
ST   GESTAX32.xMinusLS           * Negative limit switch

LD   AXLSREF32.y_MAX_LS          * Max Limit switch
ST   GESTAX32.xPlusLS            * Positive limit switch

LD   AXLSREF32.y_REF_S           * Reference switch
ST   GESTAX32.xRefLS             * Reference
***

LD   TON_ABIL.Q          * Abilitazione drives
ANDN TOF_MALARM.Q        * Assi in allarme
AND  Pon                           ** PON
ST   GESTAX32.xCloseLoop

LD   GSTMAC.yChSelMask.3
AND  SEL_ASSE.yExtMask.6
ST   GESTAX32.xSelected

***************************************
* Change REF quota for ABS reference
***************************************
CAL  RTRIG_AX_SEL32(CLK:=GESTAX32.xSelected)
LD   RTRIG_AX_SEL32.Q
JMPCN NoSel32
LD   ActualQtaAbsRef               ** Absolute homing quota
ST   QtaRefAbsSet                  ** Absolute homing quota setting
NoSel32:

LD   GESTAX32.xSelected
AND  %nvel14.0                     * Se Vale 1 ?gestito "Encoder Assoluto" (Da Configura Asse)
AND (
LD   ActualQtaAbsRef               ** Absolute homing quota
NE   QtaRefAbsSet                  ** Absolute homing quota setting
)
JMPCN NoEq32

LD   QtaRefAbsSet                  ** Absolute homing quota setting
ST   ActualQtaAbsRef               ** Absolute homing quota
NoEq32:
***************************************

LD   Pul_Jogp                      ** (gPlc0.4)jog+ pushbutton
AND  EnabJogRTCP                   ** Abilita Jog RTCP
ANDN EMER_GEN                      ** M0.10 Emergenza generale
AND  GESTAX32.xSelected
AND  GESTAX32.xCloseLoop
ST   GESTAX32.xJogPlus

LD   Pul_Jogm                      ** (gPlc0.5)jog- pushbutton
AND  EnabJogRTCP                   ** Abilita Jog RTCP
ANDN EMER_GEN                      ** M0.10 Emergenza generale
AND  GESTAX32.xSelected
AND  GESTAX32.xCloseLoop
ST   GESTAX32.xJogMinus

LD   %nvel14.0                     * Se Vale 1 ?gestito "Encoder Assoluto" (Da Configura Asse)
ST   GESTAX32.xZeroForced          * Forzamento asse tarato

LD   AxesHeadNoZeroed              ** Assi Testa non riferiti
OR   BlcAvX1_user                  ** M74.0 Blocco avanzamento asse X1 da user.plc
OR   BlcAvY1_user                  ** M74.4 Blocco avanzamento asse Y da user.plc
OR   CMD_HOLDMOVING_CH3.6          ** M202 Hold moving command axis CH3 (bit0=X, bit1=Y...)
ST   GESTAX32.xHoldMoving          * Richiesta blocco avanzamento

LD   Res_Axes                      ** (gPlc25.1) reset axes disable electric shaft
ST   GESTAX32.xUnlock

LDN  ch3_in_ref                    ** channel 3 in ref
ANDN EnJogRtcp                     ** (gPlc0.18)Abilitazione Jog RTCP tuning
ST   GESTAX32.xEnFIR               * Abilita filtri FIR
ST   GESTAX32.xEnFrComp            ** Abilita friction compensation

LD   ALWAYS_ZERO                   ** PLCFLAGS.0  Flag sempre stato off
ST   GESTAX32.xDisLimiter

LD   %cn0.rc8.3            * ch0 in alarm
OR   %cn3.rc8.3            * ch3 in alarm
OR   EmerINC
ST   GESTAX32.xSetAlarm     ** Forzamento allarme asse

CAL  GESTAX32

LD   JOGrunning                    ** One axis moving in JOG
OR   %ra19.1         * Stato JOG all'interno del canale
ST   JOGrunning                    ** One axis moving in JOG

LD   REFrunning                    ** One axis moving in REF
OR   %ra19.2
ST   REFrunning                    ** One axis moving in REF

LD   INCrunning                    ** One axis moving in INC
OR   %ra19.3
ST   INCrunning                    ** One axis moving in INC

LD   GESTAX32.yDriveNotEn
S    %PLCerr2.9          * Axis 32, drive not enable

LD   %pa9                * Velocit?massima asse
MUL  1000
DIV  60
ST   %ra50               * Limitazione velocita' massima interpolazione

LD   BSG_INC                       ** rg1.2 Selezione modo INC (inc.fissi)
JMPCN SVIX32

LD   %pa59               * Velocit?di Repos
MUL  1000
DIV  60
MUL  AxesOverride                  ** (gPlc16) feed degli assi (%)
DIV  100
ST   %ra50               * Limitazione velocita' massima interpolazione

SVIX32:
NOAX32:

*******************************************************************************
*   HEAD1: B (33) axis
*******************************************************************************
PATH %ax33
PATH %ax_lsref33

***************************************
*   POWER ON (PON)
***************************************
LD   %pa3.31            * Simulato
ORN  %cn3.cc1.7         * Maschera assi associata al canale
OR(
LD   %nvel11            ** 1=Mechatrolink
EQ   1
AND  %ring.drv1.RDD_wStatus.4 * PON
)
OR(
LD   %nvel11            ** 3,4=CANopen, Ecat
EQ   3
)
OR(
LD   %nvel11            ** 3,4=CANopen, Ecat
EQ   4
)
OR   (
LD   I_I_READY_DRIVE_B             ** Ready signal drive B
AND  (
LD   %ax9.nvel11
EQ   0
)
)
ST   Pon_B                         ** PON Axe B

LD  %cn3.cc1.7           * Maschera assi associata al canale 0
JMPCN NOAX33

***
*   LIMIT SWITCH & REFERENCE SWITCH

LD   %lsrefmode
ST   AXLSREF33.x_REF_mode        * 0=use ref switch...

LD   %lsreflevel
ST   AXLSREF33.x_TYPE_LS         * (1=NC, 0=NO)

LD   I_I_FC_B1_NEG                 ** B1 minimumm limit switch
ST   AXLSREF33.x_MIN_LS          * Min Limit switch

LD   I_I_FC_B1_POS                 ** B1 maximun limit switch
ST   AXLSREF33.x_MAX_LS          * Max Limit switch

LD   I_I_INDEX_B1                  ** B1 Axis Homing Switch
ST   AXLSREF33.x_REF_S           * Reference switch

CAL  AXLSREF33

LD   AXLSREF33.y_MIN_LS          * Min Limit switch
ST   GESTAX33.xMinusLS           * Negative limit switch

LD   AXLSREF33.y_MAX_LS          * Max Limit switch
ST   GESTAX33.xPlusLS            * Positive limit switch

LD   AXLSREF33.y_REF_S           * Reference switch
ST   GESTAX33.xRefLS             * Reference
***

LD   TON_ABIL.Q          * Abilitazione drives
ANDN TOF_MALARM.Q        * Assi in allarme
AND  Pon                           ** PON
ST   GESTAX33.xCloseLoop
